  MoveL 6800 to (459.4, 541.64, 120) mm, rotated rx -180 ry 0 rz 160 deg; joints [12.499, 54.474, 8.674, -144.472, 67.608, 164.783]
  Set speed (16.1 mm/s)
  Call Extruder(646.01454)
  MoveL 6801 to (458.56, 540.8, 120) mm, rotated rx 180 ry 0 rz 160 deg; joints [12.412, 54.338, 8.962, -144.599, 67.708, 164.913]
  Set speed (16.1 mm/s)
  Call Extruder(649.31213)
  MoveL 6802 to (457.9, 540.12, 120) mm, rotated rx 180 ry 0 rz 160 deg; joints [12.341, 54.231, 9.187, -144.701, 67.786, 165.015]
  Set speed (16.1 mm/s)
  Call Extruder(654.34970)
  MoveL 6803 to (456.92, 539.07, 120) mm, rotated rx 180 ry 0 rz 160 deg; joints [12.227, 54.071, 9.524, -144.861, 67.902, 165.17]
  Set speed (16.1 mm/s)
  Call Extruder(658.51823)
  MoveL 6804 to (456.13, 538.18, 120) mm, rotated rx 180 ry 0 rz 160 deg; joints [12.13, 53.942, 9.797, -144.996, 67.995, 165.297]
  Set speed (16.1 mm/s)
  Call Extruder(662.65319)
  MoveL 6805 to (455.36, 537.28, 120) mm, rotated rx 180 ry 0 rz 160 deg; joints [12.031, 53.815, 10.064, -145.132, 68.085, 165.422]
  Set speed (16.1 mm/s)
  Call Extruder(666.83023)
  MoveL 6806 to (454.61, 536.36, 120) mm, rotated rx -180 ry 0 rz 160 deg; joints [11.927, 53.691, 10.328, -145.272, 68.173, 165.548]
  Call Extruder(670.95263)
  MoveL 6807 to (453.88, 535.43, 120) mm, rotated rx 180 ry 0 rz 160 deg; joints [11.822, 53.57, 10.582, -145.412, 68.257, 165.671]
  Set speed (16.1 mm/s)
  Call Extruder(675.12873)
  MoveL 6808 to (453.16, 534.48, 120) mm, rotated rx 180 ry 0 rz 160 deg; joints [11.713, 53.451, 10.836, -145.556, 68.34, 165.795]
  Set speed (16.1 mm/s)
  Call Extruder(679.32869)
  MoveL 6809 to (452.46, 533.5, 120) mm, rotated rx 180 ry 0 rz 160 deg; joints [11.599, 53.333, 11.084, -145.704, 68.421, 165.918]
  Set speed (16.1 mm/s)
  Call Extruder(683.43317)
  MoveL 6810 to (451.8, 532.54, 120) mm, rotated rx -180 ry 0 rz 160 deg; joints [11.485, 53.221, 11.321, -145.851, 68.497, 166.037]
  Set speed (16.1 mm/s)
  Call Extruder(686.86357)
  MoveL 6811 to (451.25, 531.72, 120) mm, rotated rx 180 ry 0 rz 160 deg; joints [11.388, 53.13, 11.516, -145.975, 68.558, 166.136]
  Set speed (16.1 mm/s)
  Call Extruder(691.76365)
  MoveL 6812 to (450.5, 530.53, 120) mm, rotated rx -180 ry 0 rz 160 deg; joints [11.246, 53.002, 11.786, -146.154, 68.643, 166.276]
  Set speed (16.1 mm/s)
  Call Extruder(695.89083)
  MoveL 6813 to (449.89, 529.52, 120) mm, rotated rx -180 ry 0 rz 160 deg; joints [11.123, 52.898, 12.007, -146.308, 68.711, 166.393]
  Set speed (16.1 mm/s)
  Call Extruder(700.22200)
  MoveL 6814 to (449.28, 528.45, 120) mm, rotated rx -180 ry 0 rz 160 deg; joints [10.991, 52.792, 12.233, -146.471, 68.78, 166.513]
  Set speed (16.1 mm/s)
  Call Extruder(704.20056)
  MoveL 6815 to (448.73, 527.46, 120) mm, rotated rx 180 ry 0 rz 160 deg; joints [10.868, 52.697, 12.434, -146.623, 68.84, 166.623]
  Set speed (16.1 mm/s)
  Call Extruder(708.45243)
  MoveL 6816 to (448.17, 526.38, 120) mm, rotated rx 180 ry 0 rz 160 deg; joints [10.733, 52.599, 12.643, -146.787, 68.902, 166.739]
  Set speed (16.1 mm/s)
  Call Extruder(712.70917)
  MoveL 6817 to (447.63, 525.29, 120) mm, rotated rx 180 ry 0 rz 160 deg; joints [10.595, 52.504, 12.846, -146.953, 68.961, 166.853]
  Call Extruder(720.90812)
  MoveL 6818 to (446.65, 523.16, 120) mm, rotated rx -180 ry 0 rz 160 deg; joints [10.323, 52.329, 13.218, -147.278, 69.065, 167.07]
  Set speed (16.1 mm/s)
  Call Extruder(729.11713)
  MoveL 6819 to (445.76, 520.99, 120) mm, rotated rx -180 ry 0 rz 160 deg; joints [10.041, 52.167, 13.564, -147.611, 69.157, 167.281]
  Set speed (16.1 mm/s)
  Call Extruder(733.49814)
  MoveL 6820 to (445.33, 519.82, 120) mm, rotated rx 180 ry 0 rz 160 deg; joints [9.886, 52.086, 13.737, -147.79, 69.201, 167.391]
  Call Extruder(737.53315)
  MoveL 6821 to (444.94, 518.73, 120) mm, rotated rx 180 ry 0 rz 160 deg; joints [9.743, 52.014, 13.892, -147.957, 69.24, 167.491]
  Set speed (16.1 mm/s)
  Call Extruder(741.86367)
  MoveL 6822 to (444.56, 517.56, 120) mm, rotated rx 180 ry 0 rz 160 deg; joints [9.586, 51.94, 14.049, -148.138, 69.277, 167.596]
  Call Extruder(745.89010)
  MoveL 6823 to (444.22, 516.46, 120) mm, rotated rx 180 ry 0 rz 160 deg; joints [9.439, 51.874, 14.191, -148.306, 69.309, 167.693]
  Set speed (16.1 mm/s)
  Call Extruder(754.18387)
  MoveL 6824 to (443.6, 514.17, 120) mm, rotated rx -180 ry 0 rz 160 deg; joints [9.129, 51.748, 14.459, -148.658, 69.366, 167.887]
  Set speed (16.1 mm/s)
  Call Extruder(757.85337)
  MoveL 6825 to (443.35, 513.15, 120) mm, rotated rx -180 ry 0 rz 160 deg; joints [8.989, 51.698, 14.568, -148.815, 69.386, 167.971]
  Set speed (16.1 mm/s)
  Call Extruder(763.31257)
  MoveL 6826 to (443.02, 511.63, 120) mm, rotated rx -180 ry 0 rz 160 deg; joints [8.78, 51.626, 14.722, -149.05, 69.413, 168.093]
  Set speed (16.1 mm/s)
  Call Extruder(771.04723)
  MoveL 6827 to (442.62, 509.46, 120) mm, rotated rx -180 ry 0 rz 160 deg; joints [8.478, 51.534, 14.918, -149.385, 69.441, 168.261]
  Set speed (16.1 mm/s)
  Call Extruder(779.38114)
  MoveL 6828 to (442.28, 507.1, 120) mm, rotated rx -180 ry 0 rz 160 deg; joints [8.148, 51.449, 15.102, -149.75, 69.459, 168.435]
  Call Extruder(787.70369)
  MoveL 6829 to (442.04, 504.74, 120) mm, rotated rx 180 ry 0 rz 160 deg; joints [7.813, 51.377, 15.255, -150.116, 69.463, 168.602]
  Call Extruder(795.81403)
  MoveL 6830 to (441.89, 502.42, 120) mm, rotated rx 180 ry 0 rz 160 deg; joints [7.483, 51.32, 15.377, -150.473, 69.455, 168.758]
  Call Extruder(804.25342)
  MoveL 6831 to (441.84, 500.01, 120) mm, rotated rx -180 ry 0 rz 160 deg; joints [7.136, 51.275, 15.474, -150.846, 69.433, 168.912]
  Set speed (16.1 mm/s)
  Call Extruder(811.82598)
  MoveL 6832 to (441.88, 497.85, 120) mm, rotated rx 180 ry 0 rz 160 deg; joints [6.823, 51.247, 15.534, -151.18, 69.401, 169.044]
  Call Extruder(819.14286)
  MoveL 6833 to (442, 495.76, 120) mm, rotated rx -180 ry 0 rz 160 deg; joints [6.52, 51.231, 15.568, -151.502, 69.36, 169.166]
  Call Extruder(826.71033)
  MoveL 6834 to (442.19, 493.61, 120) mm, rotated rx 180 ry 0 rz 160 deg; joints [6.205, 51.226, 15.58, -151.833, 69.307, 169.286]
  Set speed (16.1 mm/s)
  Call Extruder(834.19803)
  MoveL 6835 to (442.47, 491.48, 120) mm, rotated rx 180 ry 0 rz 160 deg; joints [5.894, 51.232, 15.566, -152.159, 69.242, 169.398]
  Call Extruder(841.79303)
  MoveL 6836 to (442.83, 489.34, 120) mm, rotated rx -180 ry 0 rz 160 deg; joints [5.578, 51.25, 15.528, -152.487, 69.167, 169.505]
  Set speed (16.1 mm/s)
  Call Extruder(849.45555)
  MoveL 6837 to (443.27, 487.19, 120) mm, rotated rx 180 ry 0 rz 160 deg; joints [5.262, 51.28, 15.464, -152.814, 69.079, 169.607]
  Call Extruder(856.66940)
  MoveL 6838 to (443.76, 485.19, 120) mm, rotated rx 180 ry 0 rz 160 deg; joints [4.966, 51.319, 15.381, -153.119, 68.986, 169.697]
  Set speed (16.1 mm/s)
  Call Extruder(864.15213)
  MoveL 6839 to (444.34, 483.13, 120) mm, rotated rx 180 ry 0 rz 160 deg; joints [4.661, 51.37, 15.27, -153.43, 68.879, 169.784]
  Set speed (16.1 mm/s)
  Call Extruder(871.56534)
  MoveL 6840 to (444.99, 481.12, 120) mm, rotated rx -180 ry 0 rz 160 deg; joints [4.362, 51.432, 15.137, -153.733, 68.763, 169.864]
  Set speed (16.1 mm/s)
  Call Extruder(879.13739)
  MoveL 6841 to (445.73, 479.08, 120) mm, rotated rx -180 ry 0 rz 160 deg; joints [4.06, 51.506, 14.978, -154.037, 68.633, 169.94]
  Set speed (16.1 mm/s)
  Call Extruder(885.78650)
  MoveL 6842 to (446.45, 477.32, 120) mm, rotated rx 180 ry 0 rz 160 deg; joints [3.799, 51.581, 14.818, -154.299, 68.511, 170.001]
  Call Extruder(894.03037)
  MoveL 6843 to (447.41, 475.17, 120) mm, rotated rx 180 ry 0 rz 160 deg; joints [3.481, 51.686, 14.593, -154.616, 68.348, 170.069]
  Set speed (16.1 mm/s)
  Call Extruder(901.71326)
  MoveL 6844 to (448.39, 473.2, 120) mm, rotated rx -180 ry 0 rz 160 deg; joints [3.19, 51.795, 14.359, -154.903, 68.185, 170.127]
  Set speed (16.1 mm/s)
  Call Extruder(909.01008)
  MoveL 6845 to (449.38, 471.37, 120) mm, rotated rx 180 ry 0 rz 160 deg; joints [2.919, 51.909, 14.115, -155.168, 68.021, 170.175]
  Set speed (16.1 mm/s)
  Call Extruder(916.69414)
  MoveL 6846 to (450.49, 469.48, 120) mm, rotated rx 180 ry 0 rz 160 deg; joints [2.64, 52.04, 13.835, -155.439, 67.838, 170.219]
  Call Extruder(924.08438)
  MoveL 6847 to (451.64, 467.7, 120) mm, rotated rx 180 ry 0 rz 160 deg; joints [2.379, 52.177, 13.544, -155.691, 67.653, 170.255]
  Set speed (16.1 mm/s)
  Call Extruder(931.57807)
  MoveL 6848 to (452.86, 465.94, 120) mm, rotated rx 180 ry 0 rz 160 deg; joints [2.122, 52.325, 13.227, -155.937, 67.456, 170.285]
  Call Extruder(939.16479)
  MoveL 6849 to (454.16, 464.21, 120) mm, rotated rx -180 ry 0 rz 160 deg; joints [1.869, 52.486, 12.884, -156.177, 67.247, 170.309]
  Set speed (16.1 mm/s)
  Call Extruder(946.56366)
  MoveL 6850 to (455.49, 462.57, 120) mm, rotated rx 180 ry 0 rz 160 deg; joints [1.631, 52.652, 12.53, -156.4, 67.035, 170.326]
  Call Extruder(954.04593)
  MoveL 6851 to (456.9, 460.96, 120) mm, rotated rx 180 ry 0 rz 160 deg; joints [1.398, 52.831, 12.151, -156.615, 66.812, 170.337]
  Set speed (16.1 mm/s)
  Call Extruder(961.81892)
  MoveL 6852 to (458.42, 459.34, 120) mm, rotated rx -180 ry 0 rz 160 deg; joints [1.166, 53.026, 11.737, -156.827, 66.571, 170.341]
  Call Extruder(968.91322)
  MoveL 6853 to (459.87, 457.91, 120) mm, rotated rx 180 ry 0 rz 160 deg; joints [0.962, 53.212, 11.341, -157.01, 66.344, 170.339]
  Call Extruder(976.52373)
  MoveL 6854 to (461.47, 456.44, 120) mm, rotated rx 180 ry 0 rz 160 deg; joints [0.753, 53.422, 10.897, -157.195, 66.093, 170.33]
  Set speed (16.1 mm/s)
  Call Extruder(984.09802)
  MoveL 6855 to (463.12, 455.04, 120) mm, rotated rx -180 ry 0 rz 160 deg; joints [0.555, 53.639, 10.437, -157.367, 65.836, 170.315]
  Set speed (16.1 mm/s)
  Call Extruder(991.96002)
  MoveL 6856 to (464.88, 453.64, 120) mm, rotated rx 180 ry 0 rz 160 deg; joints [0.36, 53.874, 9.94, -157.533, 65.562, 170.291]
  Call Extruder(999.08695)
  MoveL 6857 to (466.52, 452.44, 120) mm, rotated rx -180 ry 0 rz 160 deg; joints [0.193, 54.095, 9.474, -157.671, 65.306, 170.264]
  Set speed (16.1 mm/s)
  Call Extruder(1006.48210)
  MoveL 6858 to (468.27, 451.26, 120) mm, rotated rx 180 ry 0 rz 160 deg; joints [0.03, 54.332, 8.974, -157.802, 65.036, 170.229]
  Set speed (16.1 mm/s)
  Call Extruder(1014.06845)
  MoveL 6859 to (470.11, 450.11, 120) mm, rotated rx 180 ry 0 rz 160 deg; joints [-0.127, 54.583, 8.445, -157.924, 64.752, 170.186]
  Set speed (16.1 mm/s)
  Call Extruder(1021.55574)
  MoveL 6860 to (471.97, 449.04, 120) mm, rotated rx 180 ry 0 rz 160 deg; joints [-0.272, 54.838, 7.909, -158.032, 64.466, 170.136]
  Set speed (16.1 mm/s)
  Call Extruder(1029.94377)
  MoveL 6861 to (474.09, 447.93, 120) mm, rotated rx 180 ry 0 rz 160 deg; joints [-0.421, 55.133, 7.291, -158.137, 64.14, 170.073]
  Set speed (16.1 mm/s)
  Call Extruder(1036.55206)
  MoveL 6862 to (475.8, 447.12, 120) mm, rotated rx 180 ry 0 rz 160 deg; joints [-0.529, 55.371, 6.791, -158.207, 63.879, 170.017]
  Set speed (16.1 mm/s)
  Call Extruder(1044.03826)
  MoveL 6863 to (477.76, 446.27, 120) mm, rotated rx -180 ry 0 rz 160 deg; joints [-0.641, 55.647, 6.213, -158.275, 63.579, 169.946]
  Set speed (16.1 mm/s)
  Call Extruder(1051.32870)
  MoveL 6864 to (479.69, 445.5, 120) mm, rotated rx -180 ry 0 rz 160 deg; joints [-0.74, 55.923, 5.638, -158.329, 63.283, 169.871]
  Call Extruder(1059.02695)
  MoveL 6865 to (481.77, 444.77, 120) mm, rotated rx -180 ry 0 rz 160 deg; joints [-0.833, 56.219, 5.018, -158.371, 62.967, 169.784]
  Call Extruder(1066.47364)
  MoveL 6866 to (483.8, 444.14, 120) mm, rotated rx 180 ry 0 rz 160 deg; joints [-0.913, 56.512, 4.407, -158.399, 62.657, 169.693]
  Call Extruder(1073.74383)
  MoveL 6867 to (485.81, 443.6, 120) mm, rotated rx -180 ry 0 rz 160 deg; joints [-0.98, 56.804, 3.801, -158.413, 62.352, 169.596]
  Set speed (16.1 mm/s)
  Call Extruder(1081.50301)
  MoveL 6868 to (487.97, 443.1, 120) mm, rotated rx 180 ry 0 rz 160 deg; joints [-1.04, 57.12, 3.144, -158.414, 62.024, 169.486]
  Call Extruder(1088.89317)
  MoveL 6869 to (490.05, 442.7, 120) mm, rotated rx 180 ry 0 rz 160 deg; joints [-1.088, 57.426, 2.51, -158.403, 61.71, 169.374]
  Set speed (16.1 mm/s)
  Call Extruder(1096.03300)
  MoveL 6870 to (492.06, 442.39, 120) mm, rotated rx -180 ry 0 rz 160 deg; joints [-1.124, 57.725, 1.889, -158.379, 61.405, 169.258]
  Set speed (16.1 mm/s)
  Call Extruder(1103.71272)
  MoveL 6871 to (494.24, 442.13, 120) mm, rotated rx 180 ry 0 rz 160 deg; joints [-1.151, 58.051, 1.214, -158.339, 61.075, 169.126]
  Set speed (16.1 mm/s)
  Call Extruder(1111.28299)
  MoveL 6872 to (496.4, 441.95, 120) mm, rotated rx 180 ry 0 rz 160 deg; joints [-1.168, 58.377, 0.541, -158.286, 60.749, 168.989]
  Set speed (16.1 mm/s)
  Call Extruder(1118.95323)
  MoveL 6873 to (498.59, 441.86, 120) mm, rotated rx -180 ry 0 rz 160 deg; joints [-1.175, 58.71, -0.147, -158.22, 60.419, 168.842]
  Set speed (16.1 mm/s)
  Call Extruder(1126.35629)
  MoveL 6874 to (500.71, 441.85, 120) mm, rotated rx -180 ry 0 rz 160 deg; joints [-1.171, 59.035, -0.816, -158.142, 60.1, 168.692]
  Call Extruder(1133.91680)
  MoveL 6875 to (502.87, 441.91, 120) mm, rotated rx -180 ry 0 rz 160 deg; joints [-1.157, 59.369, -1.504, -158.05, 59.774, 168.532]
  Call Extruder(1141.32935)
  MoveL 6876 to (504.98, 442.06, 120) mm, rotated rx 180 ry 0 rz 160 deg; joints [-1.133, 59.699, -2.182, -157.947, 59.456, 168.367]
  Set speed (16.1 mm/s)
  Call Extruder(1148.64149)
  MoveL 6877 to (507.06, 442.27, 120) mm, rotated rx -180 ry 0 rz 160 deg; joints [-1.101, 60.026, -2.853, -157.833, 59.144, 168.197]
  Set speed (16.1 mm/s)
  Call Extruder(1156.31820)
  MoveL 6878 to (509.23, 442.58, 120) mm, rotated rx -180 ry 0 rz 160 deg; joints [-1.057, 60.371, -3.56, -157.701, 58.818, 168.012]
  Set speed (16.1 mm/s)
  Call Extruder(1163.87434)
  MoveL 6879 to (511.36, 442.96, 120) mm, rotated rx 180 ry 0 rz 160 deg; joints [-1.005, 60.711, -4.256, -157.559, 58.5, 167.822]
  Set speed (16.1 mm/s)
  Call Extruder(1171.29769)
  MoveL 6880 to (513.43, 443.41, 120) mm, rotated rx 180 ry 0 rz 160 deg; joints [-0.945, 61.046, -4.941, -157.407, 58.189, 167.628]
  Set speed (16.1 mm/s)
  Call Extruder(1178.67571)
  MoveL 6881 to (515.47, 443.94, 120) mm, rotated rx -180 ry 0 rz 160 deg; joints [-0.876, 61.38, -5.622, -157.244, 57.884, 167.429]
  Set speed (16.1 mm/s)
  Call Extruder(1186.11275)
  MoveL 6882 to (517.51, 444.54, 120) mm, rotated rx 180 ry 0 rz 160 deg; joints [-0.798, 61.715, -6.306, -157.068, 57.58, 167.221]
  Call Extruder(1193.83773)
  MoveL 6883 to (519.6, 445.25, 120) mm, rotated rx -180 ry 0 rz 160 deg; joints [-0.708, 62.063, -7.015, -156.874, 57.268, 166.997]
  Set speed (16.1 mm/s)
  Call Extruder(1201.22298)
  MoveL 6884 to (521.58, 445.99, 120) mm, rotated rx -180 ry 0 rz 160 deg; joints [-0.614, 62.395, -7.689, -156.678, 56.974, 166.777]
  Set speed (16.1 mm/s)
  Call Extruder(1208.63995)
  MoveL 6885 to (523.53, 446.82, 120) mm, rotated rx -180 ry 0 rz 160 deg; joints [-0.512, 62.726, -8.363, -156.47, 56.683, 166.549]
  Set speed (16.1 mm/s)
  Call Extruder(1215.26606)
  MoveL 6886 to (525.25, 447.61, 120) mm, rotated rx -180 ry 0 rz 160 deg; joints [-0.414, 63.021, -8.961, -156.277, 56.428, 166.341]
  Set speed (16.1 mm/s)
  Call Extruder(1223.71389)
  MoveL 6887 to (527.4, 448.7, 120) mm, rotated rx -180 ry 0 rz 160 deg; joints [-0.281, 63.393, -9.716, -156.017, 56.11, 166.069]
  Set speed (16.1 mm/s)
  Call Extruder(1231.29077)
  MoveL 6888 to (529.3, 449.76, 120) mm, rotated rx 180 ry 0 rz 160 deg; joints [-0.153, 63.725, -10.387, -155.774, 55.831, 165.818]
  Set speed (16.1 mm/s)
  Call Extruder(1238.69731)
  MoveL 6889 to (531.11, 450.86, 120) mm, rotated rx 180 ry 0 rz 160 deg; joints [-0.022, 64.045, -11.035, -155.528, 55.565, 165.567]
  Set speed (16.1 mm/s)
  Call Extruder(1246.28249)
  MoveL 6890 to (532.92, 452.06, 120) mm, rotated rx 180 ry 0 rz 160 deg; joints [0.12, 64.369, -11.69, -155.266, 55.3, 165.305]
  Set speed (16.1 mm/s)
  Call Extruder(1253.66351)
  MoveL 6891 to (534.63, 453.28, 120) mm, rotated rx 180 ry 0 rz 160 deg; joints [0.265, 64.681, -12.319, -155.003, 55.049, 165.045]
  Call Extruder(1261.15428)
  MoveL 6892 to (536.33, 454.59, 120) mm, rotated rx 180 ry 0 rz 160 deg; joints [0.418, 64.992, -12.946, -154.728, 54.803, 164.778]
  Set speed (16.1 mm/s)
  Call Extruder(1268.66408)
  MoveL 6893 to (537.98, 455.96, 120) mm, rotated rx 180 ry 0 rz 160 deg; joints [0.578, 65.298, -13.563, -154.444, 54.564, 164.505]
  Set speed (16.1 mm/s)
  Call Extruder(1276.05790)
  MoveL 6894 to (539.55, 457.37, 120) mm, rotated rx 180 ry 0 rz 160 deg; joints [0.741, 65.594, -14.16, -154.158, 54.338, 164.233]
  Set speed (16.1 mm/s)
  Call Extruder(1283.76960)
  MoveL 6895 to (541.14, 458.9, 120) mm, rotated rx 180 ry 0 rz 160 deg; joints [0.917, 65.897, -14.768, -153.853, 54.112, 163.945]
  Call Extruder(1287.76845)
  MoveL 6896 to (541.94, 459.71, 120) mm, rotated rx 180 ry 0 rz 160 deg; joints [1.011, 66.051, -15.078, -153.692, 53.998, 163.795]
  Set speed (16.1 mm/s)
  Call Extruder(1291.96467)
  MoveL 6897 to (542.76, 460.58, 120) mm, rotated rx 180 ry 0 rz 160 deg; joints [1.111, 66.211, -15.398, -153.521, 53.882, 163.637]
  Set speed (16.1 mm/s)
  Call Extruder(1296.08175)
  MoveL 6898 to (543.55, 461.46, 120) mm, rotated rx -180 ry 0 rz 160 deg; joints [1.211, 66.364, -15.707, -153.352, 53.771, 163.481]
  Set speed (16.1 mm/s)
  Call Extruder(1300.19670)
  MoveL 6899 to (544.32, 462.35, 120) mm, rotated rx -180 ry 0 rz 160 deg; joints [1.312, 66.517, -16.012, -153.181, 53.664, 163.324]
  Set speed (16.1 mm/s)
  Call Extruder(1304.40956)
  MoveL 6900 to (545.09, 463.27, 120) mm, rotated rx 180 ry 0 rz 160 deg; joints [1.417, 66.67, -16.319, -153.005, 53.557, 163.164]
  Call Extruder(1308.57141)
  MoveL 6901 to (545.83, 464.2, 120) mm, rotated rx -180 ry 0 rz 160 deg; joints [1.522, 66.818, -16.617, -152.829, 53.454, 163.004]
  Call Extruder(1312.66863)
  MoveL 6902 to (546.55, 465.13, 120) mm, rotated rx 180 ry 0 rz 160 deg; joints [1.628, 66.962, -16.905, -152.654, 53.357, 162.847]
  Set speed (16.1 mm/s)
  Call Extruder(1316.96653)
  MoveL 6903 to (547.27, 466.12, 120) mm, rotated rx -180 ry 0 rz 160 deg; joints [1.74, 67.11, -17.202, -152.47, 53.258, 162.682]
  Call Extruder(1321.10983)
  MoveL 6904 to (547.95, 467.09, 120) mm, rotated rx 180 ry 0 rz 160 deg; joints [1.849, 67.25, -17.482, -152.291, 53.167, 162.523]
  Call Extruder(1325.92423)
  MoveL 6905 to (548.72, 468.24, 120) mm, rotated rx -180 ry 0 rz 160 deg; joints [1.978, 67.409, -17.801, -152.082, 53.064, 162.338]
  Call Extruder(1329.43388)
  MoveL 6906 to (549.26, 469.08, 120) mm, rotated rx -180 ry 0 rz 160 deg; joints [2.073, 67.522, -18.027, -151.929, 52.993, 162.203]
  Set speed (16.1 mm/s)
  Call Extruder(1333.55402)
  MoveL 6907 to (549.87, 470.09, 120) mm, rotated rx -180 ry 0 rz 160 deg; joints [2.185, 67.653, -18.288, -151.748, 52.913, 162.045]
  Set speed (16.1 mm/s)
  Call Extruder(1337.62936)
  MoveL 6908 to (550.46, 471.09, 120) mm, rotated rx -180 ry 0 rz 160 deg; joints [2.297, 67.779, -18.54, -151.569, 52.837, 161.89]
  Set speed (16.1 mm/s)
  Call Extruder(1341.78518)
  MoveL 6909 to (551.04, 472.13, 120) mm, rotated rx 180 ry 0 rz 160 deg; joints [2.413, 67.904, -18.791, -151.385, 52.763, 161.731]
  Set speed (16.1 mm/s)
  Call Extruder(1345.99468)
  MoveL 6910 to (551.61, 473.19, 120) mm, rotated rx -180 ry 0 rz 160 deg; joints [2.532, 68.028, -19.038, -151.199, 52.692, 161.571]
  Set speed (16.1 mm/s)
  Call Extruder(1350.18264)
  MoveL 6911 to (552.15, 474.26, 120) mm, rotated rx -180 ry 0 rz 160 deg; joints [2.651, 68.148, -19.277, -151.013, 52.625, 161.412]
  Set speed (16.1 mm/s)
  Call Extruder(1354.31072)
  MoveL 6912 to (552.66, 475.32, 120) mm, rotated rx 180 ry 0 rz 160 deg; joints [2.769, 68.262, -19.505, -150.829, 52.563, 161.257]
  Set speed (16.1 mm/s)
  Call Extruder(1358.53123)
  MoveL 6913 to (553.16, 476.42, 120) mm, rotated rx 180 ry 0 rz 160 deg; joints [2.891, 68.375, -19.731, -150.642, 52.504, 161.099]
  Call Extruder(1366.91580)
  MoveL 6914 to (554.09, 478.63, 120) mm, rotated rx 180 ry 0 rz 160 deg; joints [3.137, 68.59, -20.16, -150.268, 52.399, 160.787]
  Set speed (16.1 mm/s)
  Call Extruder(1375.14529)
  MoveL 6915 to (554.91, 480.83, 120) mm, rotated rx -180 ry 0 rz 160 deg; joints [3.381, 68.786, -20.55, -149.901, 52.311, 160.487]
  Set speed (16.1 mm/s)
  Call Extruder(1379.37701)
  MoveL 6916 to (555.29, 481.98, 120) mm, rotated rx 180 ry 0 rz 160 deg; joints [3.509, 68.88, -20.737, -149.714, 52.273, 160.335]
  Call Extruder(1383.73199)
  MoveL 6917 to (555.67, 483.16, 120) mm, rotated rx 180 ry 0 rz 160 deg; joints [3.64, 68.974, -20.925, -149.521, 52.237, 160.179]
  Call Extruder(1387.70261)
  MoveL 6918 to (555.98, 484.25, 120) mm, rotated rx -180 ry 0 rz 160 deg; joints [3.761, 69.054, -21.085, -149.346, 52.209, 160.04]
  Set speed (16.1 mm/s)
  Call Extruder(1391.64358)
  MoveL 6919 to (556.28, 485.34, 120) mm, rotated rx 180 ry 0 rz 160 deg; joints [3.881, 69.132, -21.24, -149.172, 52.184, 159.902]
  Set speed (16.1 mm/s)
  Call Extruder(1400.07126)
  MoveL 6920 to (556.84, 487.68, 120) mm, rotated rx 180 ry 0 rz 160 deg; joints [4.141, 69.285, -21.544, -148.803, 52.144, 159.614]
  Set speed (16.1 mm/s)
  Call Extruder(1408.49387)
  MoveL 6921 to (557.3, 490.05, 120) mm, rotated rx 180 ry 0 rz 160 deg; joints [4.403, 69.42, -21.813, -148.438, 52.122, 159.335]
  Set speed (16.1 mm/s)
  Call Extruder(1416.73608)
  MoveL 6922 to (557.65, 492.37, 120) mm, rotated rx 180 ry 0 rz 160 deg; joints [4.661, 69.535, -22.041, -148.085, 52.117, 159.072]
  Set speed (16.1 mm/s)
  Call Extruder(1425.23980)
  MoveL 6923 to (557.92, 494.79, 120) mm, rotated rx 180 ry 0 rz 160 deg; joints [4.93, 69.635, -22.242, -147.727, 52.129, 158.81]
  Set speed (16.1 mm/s)
  Call Extruder(1433.45629)
  MoveL 6924 to (558.09, 497.13, 120) mm, rotated rx -180 ry 0 rz 160 deg; joints [5.191, 69.715, -22.399, -147.386, 52.158, 158.567]
  Set speed (16.1 mm/s)
  Call Extruder(1441.77748)
  MoveL 6925 to (558.16, 499.51, 120) mm, rotated rx 180 ry 0 rz 160 deg; joints [5.456, 69.777, -22.524, -147.047, 52.203, 158.333]
  Set speed (16.1 mm/s)
  Call Extruder(1449.93682)
  MoveL 6926 to (558.13, 501.85, 120) mm, rotated rx 180 ry 0 rz 160 deg; joints [5.718, 69.821, -22.61, -146.722, 52.265, 158.116]
  Set speed (16.1 mm/s)
  Call Extruder(1458.38997)
  MoveL 6927 to (558, 504.26, 120) mm, rotated rx 180 ry 0 rz 160 deg; joints [5.989, 69.846, -22.661, -146.393, 52.345, 157.903]
  Set speed (16.1 mm/s)
  Call Extruder(1466.71982)
  MoveL 6928 to (557.78, 506.63, 120) mm, rotated rx 180 ry 0 rz 160 deg; joints [6.256, 69.853, -22.674, -146.078, 52.441, 157.708]
  Set speed (16.1 mm/s)
  Call Extruder(1475.15035)
  MoveL 6929 to (557.45, 509.02, 120) mm, rotated rx -180 ry 0 rz 160 deg; joints [6.527, 69.841, -22.65, -145.768, 52.554, 157.525]
  Set speed (16.1 mm/s)
  Call Extruder(1483.23849)
  MoveL 6930 to (557.05, 511.3, 120) mm, rotated rx -180 ry 0 rz 160 deg; joints [6.787, 69.811, -22.591, -145.479, 52.677, 157.362]
  Set speed (16.1 mm/s)
  Call Extruder(1491.85094)
  MoveL 6931 to (556.52, 513.71, 120) mm, rotated rx 180 ry 0 rz 160 deg; joints [7.062, 69.76, -22.49, -145.181, 52.825, 157.205]
  Set speed (16.1 mm/s)
  Call Extruder(1499.78968)
  MoveL 6932 to (555.94, 515.9, 120) mm, rotated rx 180 ry 0 rz 160 deg; joints [7.315, 69.696, -22.362, -144.916, 52.976, 157.074]
  Set speed (16.1 mm/s)
  Call Extruder(1508.42581)
  MoveL 6933 to (555.22, 518.26, 120) mm, rotated rx 180 ry 0 rz 160 deg; joints [7.589, 69.607, -22.185, -144.639, 53.154, 156.948]
  Set speed (16.1 mm/s)
  Call Extruder(1516.59565)
  MoveL 6934 to (554.44, 520.46, 120) mm, rotated rx 180 ry 0 rz 160 deg; joints [7.847, 69.506, -21.983, -144.387, 53.337, 156.844]
  Set speed (16.1 mm/s)
  Call Extruder(1524.82299)
  MoveL 6935 to (553.57, 522.65, 120) mm, rotated rx -180 ry 0 rz 160 deg; joints [8.104, 69.387, -21.747, -144.143, 53.534, 156.754]
  Set speed (16.1 mm/s)
  Call Extruder(1533.21607)
  MoveL 6936 to (552.59, 524.84, 120) mm, rotated rx 180 ry 0 rz 160 deg; joints [8.365, 69.247, -21.469, -143.905, 53.749, 156.678]
  Set speed (16.1 mm/s)
  Call Extruder(1537.37064)
  MoveL 6937 to (552.07, 525.91, 120) mm, rotated rx -180 ry 0 rz 160 deg; joints [8.493, 69.171, -21.318, -143.792, 53.86, 156.647]
  Set speed (16.1 mm/s)
  Call Extruder(1543.51098)
  MoveL 6938 to (551.26, 527.47, 120) mm, rotated rx 180 ry 0 rz 160 deg; joints [8.681, 69.053, -21.083, -143.629, 54.029, 156.607]
  Set speed (16.2 mm/s)
  Call Extruder(1549.80649)
  MoveL 6939 to (550.39, 529.04, 120) mm, rotated rx 180 ry 0 rz 160 deg; joints [8.873, 68.921, -20.821, -143.468, 54.211, 156.576]
  Set speed (16.1 mm/s)
  Call Extruder(1553.96982)
  MoveL 6940 to (549.78, 530.07, 120) mm, rotated rx -180 ry 0 rz 160 deg; joints [8.998, 68.83, -20.639, -143.365, 54.333, 156.56]
  Call Extruder(1558.22289)
  MoveL 6941 to (549.14, 531.1, 120) mm, rotated rx -180 ry 0 rz 160 deg; joints [9.125, 68.732, -20.443, -143.264, 54.462, 156.548]
  Set speed (16.1 mm/s)
  Call Extruder(1562.31252)
  MoveL 6942 to (548.51, 532.09, 120) mm, rotated rx 180 ry 0 rz 160 deg; joints [9.247, 68.635, -20.249, -143.168, 54.588, 156.54]
  Set speed (16.1 mm/s)
  Call Extruder(1566.58984)
  MoveL 6943 to (547.82, 533.1, 120) mm, rotated rx 180 ry 0 rz 160 deg; joints [9.373, 68.529, -20.038, -143.071, 54.722, 156.535]
  Set speed (16.1 mm/s)
  Call Extruder(1571.39278)
  MoveL 6944 to (547.02, 534.22, 120) mm, rotated rx -180 ry 0 rz 160 deg; joints [9.513, 68.405, -19.79, -142.966, 54.877, 156.535]
  Call Extruder(0.00000)
  Call Extruder(3.43739)
  MoveL 6945 to (546.44, 535.01, 120) mm, rotated rx 180 ry 0 rz 160 deg; joints [9.613, 68.314, -19.609, -142.892, 54.989, 156.537]
  Set speed (16.1 mm/s)
  Call Extruder(8.16081)
  MoveL 6946 to (545.62, 536.08, 120) mm, rotated rx -180 ry 0 rz 160 deg; joints [9.749, 68.185, -19.351, -142.794, 55.146, 156.545]
  Set speed (16.1 mm/s)
  Call Extruder(11.80532)
  MoveL 6947 to (544.96, 536.89, 120) mm, rotated rx 180 ry 0 rz 160 deg; joints [9.853, 68.082, -19.145, -142.721, 55.269, 156.554]
  Set speed (16.1 mm/s)
  Call Extruder(15.90025)
  MoveL 6948 to (544.21, 537.78, 120) mm, rotated rx 180 ry 0 rz 160 deg; joints [9.969, 67.963, -18.907, -142.642, 55.409, 156.569]
  Set speed (16.1 mm/s)
  Call Extruder(20.03659)
  MoveL 6949 to (543.43, 538.68, 120) mm, rotated rx 180 ry 0 rz 160 deg; joints [10.085, 67.839, -18.661, -142.564, 55.553, 156.586]
  Set speed (16.1 mm/s)
  Call Extruder(24.30870)
  MoveL 6950 to (542.61, 539.58, 120) mm, rotated rx -180 ry 0 rz 160 deg; joints [10.204, 67.709, -18.4, -142.487, 55.704, 156.608]
  Set speed (16.1 mm/s)
  Call Extruder(28.36774)
  MoveL 6951 to (541.81, 540.42, 120) mm, rotated rx 180 ry 0 rz 160 deg; joints [10.315, 67.581, -18.145, -142.416, 55.849, 156.632]
  Set speed (16.1 mm/s)
  Call Extruder(32.58030)
  MoveL 6952 to (540.97, 541.28, 120) mm, rotated rx -180 ry 0 rz 160 deg; joints [10.429, 67.446, -17.875, -142.345, 56.001, 156.661]
  Set speed (16.1 mm/s)
  Call Extruder(36.77160)
  MoveL 6953 to (540.11, 542.12, 120) mm, rotated rx 180 ry 0 rz 160 deg; joints [10.542, 67.309, -17.601, -142.277, 56.155, 156.692]
  Set speed (16.1 mm/s)
  Call Extruder(40.84066)
  MoveL 6954 to (539.26, 542.91, 120) mm, rotated rx -180 ry 0 rz 160 deg; joints [10.65, 67.173, -17.328, -142.214, 56.305, 156.727]
  Set speed (16.1 mm/s)
  Call Extruder(44.99678)
  MoveL 6955 to (538.37, 543.7, 120) mm, rotated rx 180 ry 0 rz 160 deg; joints [10.758, 67.031, -17.043, -142.151, 56.461, 156.765]
  Set speed (16.1 mm/s)
  Call Extruder(49.25698)
  MoveL 6956 to (537.45, 544.49, 120) mm, rotated rx -180 ry 0 rz 160 deg; joints [10.868, 66.883, -16.746, -142.091, 56.622, 156.808]
  Set speed (16.1 mm/s)
  Call Extruder(53.34054)
  MoveL 6957 to (536.55, 545.24, 120) mm, rotated rx 180 ry 0 rz 160 deg; joints [10.973, 66.738, -16.457, -142.035, 56.777, 156.852]
  Set speed (16.1 mm/s)
  Call Extruder(57.63629)
  MoveL 6958 to (535.59, 546, 120) mm, rotated rx -180 ry 0 rz 160 deg; joints [11.081, 66.583, -16.146, -141.979, 56.942, 156.901]
  Set speed (16.1 mm/s)
  Call Extruder(61.65074)
  MoveL 6959 to (534.67, 546.69, 120) mm, rotated rx 180 ry 0 rz 160 deg; joints [11.18, 66.436, -15.85, -141.929, 57.098, 156.951]
  Set speed (16.1 mm/s)
  Call Extruder(65.84245)
  MoveL 6960 to (533.7, 547.4, 120) mm, rotated rx 180 ry 0 rz 160 deg; joints [11.282, 66.28, -15.538, -141.879, 57.261, 157.005]
  Set speed (16.1 mm/s)
  Call Extruder(69.96501)
  MoveL 6961 to (532.74, 548.07, 120) mm, rotated rx -180 ry 0 rz 160 deg; joints [11.381, 66.124, -15.225, -141.833, 57.423, 157.062]
  Set speed (16.1 mm/s)
  Call Extruder(74.19741)
  MoveL 6962 to (531.73, 548.74, 120) mm, rotated rx 180 ry 0 rz 160 deg; joints [11.481, 65.962, -14.899, -141.789, 57.591, 157.124]
  Call Extruder(78.26454)
  MoveL 6963 to (530.75, 549.37, 120) mm, rotated rx -180 ry 0 rz 160 deg; joints [11.576, 65.805, -14.582, -141.748, 57.753, 157.185]
  Set speed (16.1 mm/s)
  Call Extruder(82.50052)
  MoveL 6964 to (529.71, 550, 120) mm, rotated rx -180 ry 0 rz 160 deg; joints [11.672, 65.638, -14.247, -141.708, 57.922, 157.252]
  Set speed (16.1 mm/s)
  Call Extruder(86.66587)
  MoveL 6965 to (528.68, 550.59, 120) mm, rotated rx 180 ry 0 rz 160 deg; joints [11.765, 65.472, -13.913, -141.672, 58.09, 157.321]
  Set speed (16.1 mm/s)
  Call Extruder(93.50570)
  MoveL 6966 to (526.97, 551.53, 120) mm, rotated rx 180 ry 0 rz 160 deg; joints [11.914, 65.197, -13.359, -141.617, 58.366, 157.44]
  Set speed (16.1 mm/s)
  Call Extruder(99.11961)
  MoveL 6967 to (525.54, 552.25, 120) mm, rotated rx -180 ry 0 rz 160 deg; joints [12.033, 64.966, -12.895, -141.579, 58.595, 157.543]
  Set speed (16.1 mm/s)
  Call Extruder(103.28725)
  MoveL 6968 to (524.46, 552.76, 120) mm, rotated rx 180 ry 0 rz 160 deg; joints [12.118, 64.794, -12.546, -141.552, 58.765, 157.623]
  Set speed (16.1 mm/s)
  Call Extruder(111.55058)
  MoveL 6969 to (522.3, 553.72, 120) mm, rotated rx 180 ry 0 rz 160 deg; joints [12.283, 64.447, -11.847, -141.507, 59.103, 157.787]
  Set speed (16.1 mm/s)
  Call Extruder(115.82777)
  MoveL 6970 to (521.16, 554.17, 120) mm, rotated rx 180 ry 0 rz 160 deg; joints [12.364, 64.265, -11.479, -141.488, 59.279, 157.877]
  Set speed (16.1 mm/s)
  Call Extruder(120.02852)
  MoveL 6971 to (520.04, 554.59, 120) mm, rotated rx -180 ry 0 rz 160 deg; joints [12.442, 64.086, -11.117, -141.471, 59.452, 157.967]
  Set speed (16.1 mm/s)
  Call Extruder(124.24046)
  MoveL 6972 to (518.91, 554.99, 120) mm, rotated rx -180 ry 0 rz 160 deg; joints [12.518, 63.904, -10.749, -141.458, 59.626, 158.06]
  Set speed (16.1 mm/s)
  Call Extruder(128.40284)
  MoveL 6973 to (517.78, 555.37, 120) mm, rotated rx -180 ry 0 rz 160 deg; joints [12.592, 63.724, -10.386, -141.446, 59.797, 158.153]
  Call Extruder(133.49486)
  MoveL 6974 to (516.39, 555.8, 120) mm, rotated rx -180 ry 0 rz 160 deg; joints [12.678, 63.502, -9.936, -141.435, 60.007, 158.27]
  Set speed (16.1 mm/s)
  Call Extruder(136.79206)
  MoveL 6975 to (515.49, 556.06, 120) mm, rotated rx 180 ry 0 rz 160 deg; joints [12.732, 63.358, -9.643, -141.43, 60.143, 158.347]
  Set speed (16.1 mm/s)
  Call Extruder(140.25398)
  MoveL 6976 to (514.53, 556.31, 120) mm, rotated rx 180 ry 0 rz 160 deg; joints [12.787, 63.205, -9.334, -141.427, 60.286, 158.431]
  Set speed (16.1 mm/s)
  Call Extruder(144.80557)
  MoveL 6977 to (513.27, 556.62, 120) mm, rotated rx -180 ry 0 rz 160 deg; joints [12.858, 63.004, -8.926, -141.425, 60.473, 158.542]
  Set speed (16.1 mm/s)
  Call Extruder(153.33811)
  MoveL 6978 to (510.88, 557.13, 120) mm, rotated rx 180 ry 0 rz 160 deg; joints [12.982, 62.624, -8.156, -141.429, 60.824, 158.756]
  Set speed (16.1 mm/s)
  Call Extruder(161.71940)
  MoveL 6979 to (508.52, 557.53, 120) mm, rotated rx -180 ry 0 rz 160 deg; joints [13.094, 62.249, -7.393, -141.443, 61.167, 158.974]
  Set speed (16.1 mm/s)
  Call Extruder(169.83564)
  MoveL 6980 to (506.22, 557.82, 120) mm, rotated rx 180 ry 0 rz 160 deg; joints [13.193, 61.884, -6.65, -141.467, 61.498, 159.192]
  Set speed (16.1 mm/s)
  Call Extruder(178.33795)
  MoveL 6981 to (503.8, 558.03, 120) mm, rotated rx -180 ry 0 rz 160 deg; joints [13.286, 61.501, -5.869, -141.502, 61.843, 159.427]
  Set speed (16.1 mm/s)
  Call Extruder(186.71052)
  MoveL 6982 to (501.41, 558.14, 120) mm, rotated rx 180 ry 0 rz 160 deg; joints [13.367, 61.122, -5.097, -141.546, 62.179, 159.664]
  Call Extruder(194.93472)
  MoveL 6983 to (499.06, 558.15, 120) mm, rotated rx -180 ry 0 rz 160 deg; joints [13.436, 60.751, -4.338, -141.599, 62.506, 159.902]
  Set speed (10.0 mm/s)
  MoveL 6984 to (499.06, 558.15, 124) mm, rotated rx -180 ry 0 rz 160 deg; joints [13.436, 60.143, -4.112, -141.475, 62.207, 159.634]
  Set speed (120.0 mm/s)
  MoveL 6985 to (499.09, 556.18, 124) mm, rotated rx 180 ry 0 rz 160 deg; joints [13.197, 60.075, -3.973, -141.752, 62.18, 159.802]
  Set speed (16.2 mm/s)
  Call Extruder(202.74859)
  MoveL 6986 to (496.86, 556.1, 124) mm, rotated rx 180 ry 0 rz 160 deg; joints [13.25, 59.72, -3.252, -141.814, 62.486, 160.032]
  Set speed (16.2 mm/s)
  Call Extruder(211.07055)
  MoveL 6987 to (494.48, 555.91, 124) mm, rotated rx 180 ry 0 rz 160 deg; joints [13.297, 59.344, -2.485, -141.89, 62.809, 160.281]
  Call Extruder(219.01827)
  MoveL 6988 to (492.22, 555.65, 124) mm, rotated rx 180 ry 0 rz 160 deg; joints [13.329, 58.986, -1.755, -141.972, 63.113, 160.522]
  Call Extruder(227.00008)
  MoveL 6989 to (489.96, 555.28, 124) mm, rotated rx 180 ry 0 rz 160 deg; joints [13.35, 58.628, -1.025, -142.065, 63.413, 160.769]
  Call Extruder(235.15992)
  MoveL 6990 to (487.67, 554.82, 124) mm, rotated rx 180 ry 0 rz 160 deg; joints [13.36, 58.266, -0.284, -142.171, 63.716, 161.024]
  Set speed (16.2 mm/s)
  Call Extruder(239.11568)
  MoveL 6991 to (486.57, 554.55, 124) mm, rotated rx -180 ry 0 rz 160 deg; joints [13.36, 58.091, 0.073, -142.226, 63.86, 161.149]
  Call Extruder(243.12891)
  MoveL 6992 to (485.45, 554.27, 124) mm, rotated rx 180 ry 0 rz 160 deg; joints [13.358, 57.915, 0.434, -142.284, 64.005, 161.276]
  Set speed (16.2 mm/s)
  Call Extruder(251.01965)
  MoveL 6993 to (483.28, 553.64, 124) mm, rotated rx 180 ry 0 rz 160 deg; joints [13.343, 57.572, 1.139, -142.406, 64.286, 161.528]
  Set speed (16.2 mm/s)
  Call Extruder(258.94151)
  MoveL 6994 to (481.13, 552.92, 124) mm, rotated rx 180 ry 0 rz 160 deg; joints [13.317, 57.23, 1.839, -142.538, 64.563, 161.782]
  Set speed (16.2 mm/s)
  Call Extruder(263.19391)
  MoveL 6995 to (479.99, 552.5, 124) mm, rotated rx -180 ry 0 rz 160 deg; joints [13.298, 57.049, 2.212, -142.614, 64.709, 161.92]
  Set speed (16.2 mm/s)
  Call Extruder(267.13807)
  MoveL 6996 to (478.93, 552.09, 124) mm, rotated rx 180 ry 0 rz 160 deg; joints [13.277, 56.882, 2.555, -142.685, 64.843, 162.047]
  Set speed (16.2 mm/s)
  Call Extruder(274.12191)
  MoveL 6997 to (477.09, 551.31, 124) mm, rotated rx -180 ry 0 rz 160 deg; joints [13.233, 56.59, 3.156, -142.819, 65.076, 162.273]
  Set speed (16.2 mm/s)
  Call Extruder(279.16492)
  MoveL 6998 to (475.78, 550.7, 124) mm, rotated rx -180 ry 0 rz 160 deg; joints [13.195, 56.382, 3.586, -142.921, 65.24, 162.437]
  Set speed (16.2 mm/s)
  Call Extruder(285.19971)
  MoveL 6999 to (474.23, 549.94, 124) mm, rotated rx -180 ry 0 rz 160 deg; joints [13.144, 56.135, 4.094, -143.048, 65.434, 162.633]
  Set speed (16.1 mm/s)
  Call Extruder(291.24257)
  MoveL 7000 to (472.71, 549.12, 124) mm, rotated rx 180 ry 0 rz 160 deg; joints [13.084, 55.892, 4.596, -143.181, 65.623, 162.83]
  Set speed (16.2 mm/s)
  Call Extruder(294.57549)
  MoveL 7001 to (471.88, 548.64, 124) mm, rotated rx 180 ry 0 rz 160 deg; joints [13.048, 55.76, 4.87, -143.257, 65.726, 162.938]
  Set speed (16.2 mm/s)
  Call Extruder(298.44787)
  MoveL 7002 to (470.93, 548.08, 124) mm, rotated rx -180 ry 0 rz 160 deg; joints [13.003, 55.607, 5.186, -143.347, 65.844, 163.064]
  Set speed (16.2 mm/s)
  Call Extruder(303.22144)
  MoveL 7003 to (469.76, 547.36, 124) mm, rotated rx 180 ry 0 rz 160 deg; joints [12.944, 55.421, 5.571, -143.462, 65.986, 163.22]
  Call Extruder(307.29979)
  MoveL 7004 to (468.79, 546.72, 124) mm, rotated rx 180 ry 0 rz 160 deg; joints [12.89, 55.264, 5.896, -143.563, 66.106, 163.352]
  Set speed (16.2 mm/s)
  Call Extruder(311.23567)
  MoveL 7005 to (467.85, 546.08, 124) mm, rotated rx -180 ry 0 rz 160 deg; joints [12.835, 55.114, 6.206, -143.663, 66.219, 163.479]
  Set speed (16.2 mm/s)
  Call Extruder(315.17150)
  MoveL 7006 to (466.93, 545.43, 124) mm, rotated rx 180 ry 0 rz 160 deg; joints [12.777, 54.967, 6.513, -143.765, 66.331, 163.606]
  Set speed (16.2 mm/s)
  Call Extruder(319.29304)
  MoveL 7007 to (465.99, 544.72, 124) mm, rotated rx -180 ry 0 rz 160 deg; joints [12.712, 54.814, 6.829, -143.876, 66.445, 163.739]
  Set speed (16.2 mm/s)
  Call Extruder(323.19809)
  MoveL 7008 to (465.1, 544.04, 124) mm, rotated rx 180 ry 0 rz 160 deg; joints [12.648, 54.671, 7.126, -143.982, 66.552, 163.865]
  Set speed (16.2 mm/s)
  Call Extruder(326.58083)
  MoveL 7009 to (464.35, 543.43, 124) mm, rotated rx -180 ry 0 rz 160 deg; joints [12.591, 54.549, 7.38, -144.076, 66.642, 163.973]
  Set speed (16.1 mm/s)
  Call Extruder(332.37087)
  MoveL 7010 to (463.08, 542.36, 124) mm, rotated rx -180 ry 0 rz 160 deg; joints [12.487, 54.344, 7.807, -144.241, 66.793, 164.158]
  Set speed (16.2 mm/s)
  Call Extruder(335.30927)
  MoveL 7011 to (462.45, 541.8, 124) mm, rotated rx 180 ry 0 rz 160 deg; joints [12.431, 54.241, 8.02, -144.326, 66.868, 164.251]
  Set speed (16.2 mm/s)
  Call Extruder(339.27302)
  MoveL 7012 to (461.62, 541.03, 124) mm, rotated rx 180 ry 0 rz 160 deg; joints [12.353, 54.105, 8.304, -144.444, 66.967, 164.376]
  Set speed (16.2 mm/s)
  Call Extruder(343.27941)
  MoveL 7013 to (460.79, 540.24, 124) mm, rotated rx 180 ry 0 rz 160 deg; joints [12.272, 53.969, 8.587, -144.566, 67.065, 164.502]
  Call Extruder(347.33894)
  MoveL 7014 to (459.96, 539.42, 124) mm, rotated rx 180 ry 0 rz 160 deg; joints [12.186, 53.834, 8.869, -144.691, 67.162, 164.629]
  Call Extruder(351.37461)
  MoveL 7015 to (459.16, 538.59, 124) mm, rotated rx -180 ry 0 rz 160 deg; joints [12.098, 53.702, 9.144, -144.819, 67.256, 164.755]
  Set speed (16.2 mm/s)
  Call Extruder(355.33922)
  MoveL 7016 to (458.39, 537.75, 124) mm, rotated rx -180 ry 0 rz 160 deg; joints [12.008, 53.575, 9.411, -144.946, 67.346, 164.878]
  Set speed (16.2 mm/s)
  Call Extruder(359.33698)
  MoveL 7017 to (457.63, 536.9, 124) mm, rotated rx 180 ry 0 rz 160 deg; joints [11.914, 53.449, 9.674, -145.077, 67.434, 165.001]
  Set speed (16.2 mm/s)
  Call Extruder(362.90095)
  MoveL 7018 to (456.96, 536.12, 124) mm, rotated rx 180 ry 0 rz 160 deg; joints [11.828, 53.338, 9.905, -145.195, 67.511, 165.109]
  Set speed (16.2 mm/s)
  Call Extruder(367.47989)
  MoveL 7019 to (456.13, 535.11, 124) mm, rotated rx 180 ry 0 rz 160 deg; joints [11.715, 53.2, 10.195, -145.35, 67.606, 165.248]
  Set speed (16.2 mm/s)
  Call Extruder(371.39933)
  MoveL 7020 to (455.44, 534.22, 124) mm, rotated rx -180 ry 0 rz 160 deg; joints [11.614, 53.083, 10.438, -145.484, 67.685, 165.366]
  Set speed (16.2 mm/s)
  Call Extruder(375.43161)
  MoveL 7021 to (454.74, 533.3, 124) mm, rotated rx -180 ry 0 rz 160 deg; joints [11.508, 52.967, 10.682, -145.625, 67.763, 165.486]
  Call Extruder(379.42273)
  MoveL 7022 to (454.08, 532.37, 124) mm, rotated rx -180 ry 0 rz 160 deg; joints [11.399, 52.854, 10.919, -145.767, 67.839, 165.605]
  Call Extruder(383.44071)
  MoveL 7023 to (453.42, 531.42, 124) mm, rotated rx -180 ry 0 rz 160 deg; joints [11.288, 52.743, 11.152, -145.912, 67.912, 165.722]
  Call Extruder(387.45535)
  MoveL 7024 to (452.79, 530.46, 124) mm, rotated rx 180 ry 0 rz 160 deg; joints [11.173, 52.634, 11.379, -146.058, 67.982, 165.839]
  Set speed (16.2 mm/s)
  Call Extruder(391.44524)
  MoveL 7025 to (452.18, 529.49, 124) mm, rotated rx 180 ry 0 rz 160 deg; joints [11.057, 52.529, 11.6, -146.206, 68.05, 165.954]
  Set speed (16.2 mm/s)
  Call Extruder(395.45767)
  MoveL 7026 to (451.58, 528.51, 124) mm, rotated rx 180 ry 0 rz 160 deg; joints [10.938, 52.427, 11.815, -146.356, 68.115, 166.068]
  Set speed (16.2 mm/s)
  Call Extruder(399.46759)
  MoveL 7027 to (451.01, 527.51, 124) mm, rotated rx 180 ry 0 rz 160 deg; joints [10.815, 52.327, 12.025, -146.508, 68.177, 166.181]
  Call Extruder(403.46596)
  MoveL 7028 to (450.46, 526.51, 124) mm, rotated rx -180 ry 0 rz 160 deg; joints [10.691, 52.23, 12.228, -146.662, 68.237, 166.293]
  Set speed (16.2 mm/s)
  Call Extruder(407.48703)
  MoveL 7029 to (449.93, 525.49, 124) mm, rotated rx 180 ry 0 rz 160 deg; joints [10.563, 52.136, 12.426, -146.818, 68.293, 166.404]
  Set speed (16.2 mm/s)
  Call Extruder(411.58177)
  MoveL 7030 to (449.4, 524.44, 124) mm, rotated rx 180 ry 0 rz 160 deg; joints [10.431, 52.043, 12.622, -146.979, 68.348, 166.515]
  Call Extruder(419.40114)
  MoveL 7031 to (448.47, 522.4, 124) mm, rotated rx 180 ry 0 rz 160 deg; joints [10.171, 51.875, 12.977, -147.291, 68.445, 166.724]
  Set speed (16.2 mm/s)
  Call Extruder(423.63458)
  MoveL 7032 to (448, 521.28, 124) mm, rotated rx 180 ry 0 rz 160 deg; joints [10.026, 51.789, 13.158, -147.463, 68.492, 166.835]
  Set speed (16.2 mm/s)
  Call Extruder(427.41496)
  MoveL 7033 to (447.6, 520.28, 124) mm, rotated rx 180 ry 0 rz 160 deg; joints [9.895, 51.714, 13.316, -147.617, 68.533, 166.933]
  Set speed (16.2 mm/s)
  Call Extruder(431.66766)
  MoveL 7034 to (447.18, 519.14, 124) mm, rotated rx -180 ry 0 rz 160 deg; joints [9.746, 51.634, 13.485, -147.793, 68.574, 167.041]
  Call Extruder(435.60722)
  MoveL 7035 to (446.8, 518.07, 124) mm, rotated rx 180 ry 0 rz 160 deg; joints [9.606, 51.562, 13.637, -147.956, 68.61, 167.141]
  Call Extruder(439.68971)
  MoveL 7036 to (446.44, 516.96, 124) mm, rotated rx 180 ry 0 rz 160 deg; joints [9.458, 51.492, 13.784, -148.127, 68.644, 167.241]
  Set speed (16.1 mm/s)
  Call Extruder(443.57911)
  MoveL 7037 to (446.11, 515.9, 124) mm, rotated rx 180 ry 0 rz 160 deg; joints [9.315, 51.427, 13.921, -148.291, 68.674, 167.336]
  Call Extruder(447.72151)
  MoveL 7038 to (445.79, 514.76, 124) mm, rotated rx -180 ry 0 rz 160 deg; joints [9.161, 51.363, 14.058, -148.467, 68.701, 167.435]
  Set speed (16.2 mm/s)
  Call Extruder(451.55459)
  MoveL 7039 to (445.51, 513.7, 124) mm, rotated rx 180 ry 0 rz 160 deg; joints [9.018, 51.305, 14.18, -148.63, 68.725, 167.526]
  Set speed (16.1 mm/s)
  Call Extruder(455.08215)
  MoveL 7040 to (445.27, 512.72, 124) mm, rotated rx 180 ry 0 rz 160 deg; joints [8.884, 51.255, 14.285, -148.782, 68.744, 167.608]
  Set speed (16.1 mm/s)
  Call Extruder(459.60503)
  MoveL 7041 to (444.99, 511.45, 124) mm, rotated rx 180 ry 0 rz 160 deg; joints [8.711, 51.194, 14.414, -148.977, 68.765, 167.711]
  Set speed (16.2 mm/s)
  Call Extruder(467.82058)
  MoveL 7042 to (444.56, 509.14, 124) mm, rotated rx 180 ry 0 rz 160 deg; joints [8.391, 51.095, 14.624, -149.334, 68.792, 167.894]
  Set speed (16.2 mm/s)
  Call Extruder(475.84535)
  MoveL 7043 to (444.24, 506.86, 124) mm, rotated rx -180 ry 0 rz 160 deg; joints [8.073, 51.012, 14.801, -149.686, 68.807, 168.065]
  Set speed (16.2 mm/s)
  Call Extruder(483.86382)
  MoveL 7044 to (444, 504.58, 124) mm, rotated rx -180 ry 0 rz 160 deg; joints [7.752, 50.941, 14.95, -150.039, 68.809, 168.229]
  Call Extruder(491.69044)
  MoveL 7045 to (443.86, 502.34, 124) mm, rotated rx 180 ry 0 rz 160 deg; joints [7.434, 50.886, 15.067, -150.385, 68.798, 168.383]
  Set speed (16.2 mm/s)
  Call Extruder(499.80493)
  MoveL 7046 to (443.81, 500.01, 124) mm, rotated rx -180 ry 0 rz 160 deg; joints [7.101, 50.842, 15.16, -150.744, 68.774, 168.535]
  Set speed (16.2 mm/s)
  Call Extruder(507.12206)
  MoveL 7047 to (443.85, 497.92, 124) mm, rotated rx 180 ry 0 rz 160 deg; joints [6.799, 50.815, 15.218, -151.067, 68.741, 168.667]
  Set speed (16.2 mm/s)
  Call Extruder(514.24372)
  MoveL 7048 to (443.96, 495.88, 124) mm, rotated rx -180 ry 0 rz 160 deg; joints [6.505, 50.799, 15.253, -151.381, 68.7, 168.789]
  Call Extruder(521.36753)
  MoveL 7049 to (444.15, 493.85, 124) mm, rotated rx 180 ry 0 rz 160 deg; joints [6.209, 50.794, 15.263, -151.693, 68.648, 168.905]
  Set speed (16.2 mm/s)
  Call Extruder(528.67979)
  MoveL 7050 to (444.42, 491.77, 124) mm, rotated rx -180 ry 0 rz 160 deg; joints [5.906, 50.8, 15.251, -152.011, 68.583, 169.018]
  Set speed (16.2 mm/s)
  Call Extruder(535.71236)
  MoveL 7051 to (444.75, 489.78, 124) mm, rotated rx 180 ry 0 rz 160 deg; joints [5.615, 50.816, 15.215, -152.315, 68.512, 169.121]
  Set speed (16.2 mm/s)
  Call Extruder(543.10448)
  MoveL 7052 to (445.18, 487.7, 124) mm, rotated rx 180 ry 0 rz 160 deg; joints [5.31, 50.845, 15.154, -152.631, 68.426, 169.223]
  Set speed (16.2 mm/s)
  Call Extruder(550.25284)
  MoveL 7053 to (445.66, 485.72, 124) mm, rotated rx 180 ry 0 rz 160 deg; joints [5.017, 50.884, 15.071, -152.932, 68.332, 169.315]
  Set speed (16.2 mm/s)
  Call Extruder(557.54745)
  MoveL 7054 to (446.23, 483.7, 124) mm, rotated rx 180 ry 0 rz 160 deg; joints [4.721, 50.935, 14.964, -153.236, 68.227, 169.404]
  Set speed (16.2 mm/s)
  Call Extruder(564.75886)
  MoveL 7055 to (446.86, 481.74, 124) mm, rotated rx 180 ry 0 rz 160 deg; joints [4.431, 50.996, 14.835, -153.531, 68.113, 169.485]
  Set speed (16.2 mm/s)
  Call Extruder(572.09248)
  MoveL 7056 to (447.59, 479.76, 124) mm, rotated rx -180 ry 0 rz 160 deg; joints [4.139, 51.069, 14.679, -153.825, 67.986, 169.561]
  Set speed (16.2 mm/s)
  Call Extruder(579.31343)
  MoveL 7057 to (448.36, 477.85, 124) mm, rotated rx 180 ry 0 rz 160 deg; joints [3.857, 51.152, 14.503, -154.108, 67.852, 169.63]
  Set speed (16.2 mm/s)
  Call Extruder(586.52203)
  MoveL 7058 to (449.21, 475.97, 124) mm, rotated rx -180 ry 0 rz 160 deg; joints [3.579, 51.246, 14.305, -154.385, 67.708, 169.693]
  Set speed (16.2 mm/s)
  Call Extruder(593.65889)
  MoveL 7059 to (450.12, 474.14, 124) mm, rotated rx -180 ry 0 rz 160 deg; joints [3.309, 51.349, 14.087, -154.652, 67.556, 169.748]
  Set speed (16.2 mm/s)
  Call Extruder(600.87426)
  MoveL 7060 to (451.11, 472.32, 124) mm, rotated rx -180 ry 0 rz 160 deg; joints [3.042, 51.463, 13.845, -154.914, 67.393, 169.799]
  Set speed (16.2 mm/s)
  Call Extruder(608.13405)
  MoveL 7061 to (452.16, 470.53, 124) mm, rotated rx -180 ry 0 rz 160 deg; joints [2.779, 51.589, 13.58, -155.17, 67.22, 169.843]
  Set speed (16.2 mm/s)
  Call Extruder(615.30930)
  MoveL 7062 to (453.27, 468.8, 124) mm, rotated rx -180 ry 0 rz 160 deg; joints [2.525, 51.723, 13.296, -155.414, 67.04, 169.881]
  Set speed (16.2 mm/s)
  Call Extruder(622.53085)
  MoveL 7063 to (454.45, 467.1, 124) mm, rotated rx -180 ry 0 rz 160 deg; joints [2.277, 51.869, 12.99, -155.652, 66.85, 169.912]
  Set speed (16.2 mm/s)
  Call Extruder(629.84455)
  MoveL 7064 to (455.71, 465.42, 124) mm, rotated rx -180 ry 0 rz 160 deg; joints [2.033, 52.026, 12.659, -155.882, 66.648, 169.937]
  Call Extruder(636.86304)
  MoveL 7065 to (456.98, 463.86, 124) mm, rotated rx -180 ry 0 rz 160 deg; joints [1.807, 52.186, 12.322, -156.094, 66.447, 169.956]
  Set speed (16.2 mm/s)
  Call Extruder(644.04649)
  MoveL 7066 to (458.33, 462.31, 124) mm, rotated rx 180 ry 0 rz 160 deg; joints [1.583, 52.359, 11.958, -156.301, 66.234, 169.968]
  Set speed (16.2 mm/s)
  Call Extruder(651.49908)
  MoveL 7067 to (459.8, 460.75, 124) mm, rotated rx 180 ry 0 rz 160 deg; joints [1.36, 52.548, 11.56, -156.504, 66.004, 169.974]
  Set speed (16.2 mm/s)
  Call Extruder(658.47929)
  MoveL 7068 to (461.22, 459.34, 124) mm, rotated rx 180 ry 0 rz 160 deg; joints [1.158, 52.734, 11.17, -156.685, 65.781, 169.974]
  Set speed (16.2 mm/s)
  Call Extruder(665.84266)
  MoveL 7069 to (462.77, 457.92, 124) mm, rotated rx 180 ry 0 rz 160 deg; joints [0.956, 52.939, 10.739, -156.864, 65.539, 169.967]
  Call Extruder(673.14817)
  MoveL 7070 to (464.37, 456.56, 124) mm, rotated rx -180 ry 0 rz 160 deg; joints [0.764, 53.152, 10.294, -157.03, 65.292, 169.953]
  Set speed (16.2 mm/s)
  Call Extruder(680.20864)
  MoveL 7071 to (465.95, 455.31, 124) mm, rotated rx 180 ry 0 rz 160 deg; joints [0.588, 53.365, 9.848, -157.179, 65.046, 169.933]
  Set speed (16.2 mm/s)
  Call Extruder(686.99149)
  MoveL 7072 to (467.52, 454.15, 124) mm, rotated rx -180 ry 0 rz 160 deg; joints [0.428, 53.578, 9.404, -157.311, 64.805, 169.908]
  Set speed (16.2 mm/s)
  Call Extruder(694.77103)
  MoveL 7073 to (469.36, 452.9, 124) mm, rotated rx -180 ry 0 rz 160 deg; joints [0.255, 53.83, 8.878, -157.45, 64.521, 169.872]
  Set speed (16.2 mm/s)
  Call Extruder(702.04307)
  MoveL 7074 to (471.13, 451.8, 124) mm, rotated rx 180 ry 0 rz 160 deg; joints [0.103, 54.073, 8.37, -157.567, 64.25, 169.832]
  Set speed (16.2 mm/s)
  Call Extruder(709.24056)
  MoveL 7075 to (472.92, 450.77, 124) mm, rotated rx -180 ry 0 rz 160 deg; joints [-0.037, 54.322, 7.852, -157.67, 63.977, 169.785]
  Call Extruder(716.42163)
  MoveL 7076 to (474.74, 449.81, 124) mm, rotated rx 180 ry 0 rz 160 deg; joints [-0.166, 54.577, 7.322, -157.761, 63.699, 169.731]
  Set speed (16.2 mm/s)
  Call Extruder(723.64601)
  MoveL 7077 to (476.6, 448.92, 124) mm, rotated rx 180 ry 0 rz 160 deg; joints [-0.286, 54.84, 6.775, -157.839, 63.415, 169.67]
  Set speed (16.2 mm/s)
  Call Extruder(730.92162)
  MoveL 7078 to (478.51, 448.08, 124) mm, rotated rx 180 ry 0 rz 160 deg; joints [-0.397, 55.112, 6.212, -157.906, 63.125, 169.602]
  Set speed (16.2 mm/s)
  Call Extruder(738.02335)
  MoveL 7079 to (480.41, 447.34, 124) mm, rotated rx 180 ry 0 rz 160 deg; joints [-0.494, 55.383, 5.65, -157.957, 62.838, 169.528]
  Set speed (16.2 mm/s)
  Call Extruder(745.28293)
  MoveL 7080 to (482.37, 446.65, 124) mm, rotated rx 180 ry 0 rz 160 deg; joints [-0.583, 55.666, 5.064, -157.997, 62.541, 169.445]
  Set speed (16.2 mm/s)
  Call Extruder(752.50876)
  MoveL 7081 to (484.35, 446.04, 124) mm, rotated rx -180 ry 0 rz 160 deg; joints [-0.662, 55.953, 4.47, -158.024, 62.242, 169.356]
  Set speed (16.2 mm/s)
  Call Extruder(759.88887)
  MoveL 7082 to (486.39, 445.49, 124) mm, rotated rx 180 ry 0 rz 160 deg; joints [-0.731, 56.252, 3.853, -158.039, 61.934, 169.258]
  Set speed (16.2 mm/s)
  Call Extruder(766.99438)
  MoveL 7083 to (488.38, 445.03, 124) mm, rotated rx -180 ry 0 rz 160 deg; joints [-0.787, 56.545, 3.25, -158.039, 61.635, 169.155]
  Set speed (16.2 mm/s)
  Call Extruder(774.04442)
  MoveL 7084 to (490.36, 444.65, 124) mm, rotated rx -180 ry 0 rz 160 deg; joints [-0.833, 56.84, 2.643, -158.027, 61.337, 169.047]
  Set speed (16.2 mm/s)
  Call Extruder(781.00031)
  MoveL 7085 to (492.33, 444.34, 124) mm, rotated rx 180 ry 0 rz 160 deg; joints [-0.87, 57.134, 2.037, -158.004, 61.042, 168.934]
  Call Extruder(788.60021)
  MoveL 7086 to (494.49, 444.09, 124) mm, rotated rx -180 ry 0 rz 160 deg; joints [-0.898, 57.46, 1.367, -157.964, 60.718, 168.802]
  Set speed (16.2 mm/s)
  Call Extruder(795.68553)
  MoveL 7087 to (496.52, 443.92, 124) mm, rotated rx 180 ry 0 rz 160 deg; joints [-0.915, 57.768, 0.737, -157.914, 60.415, 168.672]
  Set speed (16.2 mm/s)
  Call Extruder(803.09224)
  MoveL 7088 to (498.64, 443.83, 124) mm, rotated rx 180 ry 0 rz 160 deg; joints [-0.923, 58.092, 0.071, -157.85, 60.098, 168.528]
  Set speed (16.2 mm/s)
  Call Extruder(810.22205)
  MoveL 7089 to (500.68, 443.82, 124) mm, rotated rx 180 ry 0 rz 160 deg; joints [-0.92, 58.408, -0.574, -157.774, 59.793, 168.383]
  Set speed (16.2 mm/s)
  Call Extruder(817.51298)
  MoveL 7090 to (502.77, 443.88, 124) mm, rotated rx 180 ry 0 rz 160 deg; joints [-0.908, 58.733, -1.239, -157.685, 59.481, 168.226]
  Call Extruder(824.63893)
  MoveL 7091 to (504.81, 444.02, 124) mm, rotated rx -180 ry 0 rz 160 deg; joints [-0.886, 59.053, -1.892, -157.586, 59.177, 168.067]
  Set speed (16.2 mm/s)
  Call Extruder(831.67742)
  MoveL 7092 to (506.82, 444.23, 124) mm, rotated rx -180 ry 0 rz 160 deg; joints [-0.856, 59.37, -2.539, -157.475, 58.879, 167.902]
  Set speed (16.2 mm/s)
  Call Extruder(839.09787)
  MoveL 7093 to (508.92, 444.53, 124) mm, rotated rx -180 ry 0 rz 160 deg; joints [-0.815, 59.706, -3.223, -157.347, 58.566, 167.721]
  Set speed (16.2 mm/s)
  Call Extruder(846.37014)
  MoveL 7094 to (510.97, 444.89, 124) mm, rotated rx -180 ry 0 rz 160 deg; joints [-0.765, 60.036, -3.894, -157.209, 58.262, 167.537]
  Set speed (16.2 mm/s)
  Call Extruder(853.35101)
  MoveL 7095 to (512.93, 445.32, 124) mm, rotated rx 180 ry 0 rz 160 deg; joints [-0.709, 60.353, -4.538, -157.066, 57.973, 167.353]
  Set speed (16.2 mm/s)
  Call Extruder(860.72139)
  MoveL 7096 to (514.98, 445.85, 124) mm, rotated rx 180 ry 0 rz 160 deg; joints [-0.641, 60.688, -5.218, -156.903, 57.67, 167.152]
  Call Extruder(867.93932)
  MoveL 7097 to (516.96, 446.43, 124) mm, rotated rx -180 ry 0 rz 160 deg; joints [-0.566, 61.016, -5.883, -156.732, 57.377, 166.948]
  Set speed (16.2 mm/s)
  Call Extruder(875.24854)
  MoveL 7098 to (518.94, 447.11, 124) mm, rotated rx -180 ry 0 rz 160 deg; joints [-0.482, 61.346, -6.553, -156.547, 57.085, 166.735]
  Set speed (16.2 mm/s)
  Call Extruder(882.36198)
  MoveL 7099 to (520.85, 447.82, 124) mm, rotated rx -180 ry 0 rz 160 deg; joints [-0.392, 61.668, -7.203, -156.358, 56.804, 166.522]
  Call Extruder(889.66452)
  MoveL 7100 to (522.78, 448.64, 124) mm, rotated rx 180 ry 0 rz 160 deg; joints [-0.292, 61.995, -7.865, -156.152, 56.522, 166.296]
  Set speed (16.2 mm/s)
  Call Extruder(896.64056)
  MoveL 7101 to (524.59, 449.48, 124) mm, rotated rx -180 ry 0 rz 160 deg; joints [-0.189, 62.307, -8.494, -155.946, 56.256, 166.075]
  Call Extruder(903.89319)
  MoveL 7102 to (526.45, 450.43, 124) mm, rotated rx 180 ry 0 rz 160 deg; joints [-0.074, 62.628, -9.142, -155.723, 55.986, 165.839]
  Set speed (16.2 mm/s)
  Call Extruder(911.31483)
  MoveL 7103 to (528.3, 451.46, 124) mm, rotated rx -180 ry 0 rz 160 deg; joints [0.05, 62.954, -9.798, -155.484, 55.715, 165.592]
  Call Extruder(918.43060)
  MoveL 7104 to (530.05, 452.52, 124) mm, rotated rx -180 ry 0 rz 160 deg; joints [0.177, 63.263, -10.42, -155.246, 55.463, 165.35]
  Set speed (16.2 mm/s)
  Call Extruder(925.74898)
  MoveL 7105 to (531.8, 453.68, 124) mm, rotated rx -180 ry 0 rz 160 deg; joints [0.314, 63.576, -11.051, -154.993, 55.21, 165.097]
  Call Extruder(932.87143)
  MoveL 7106 to (533.46, 454.86, 124) mm, rotated rx 180 ry 0 rz 160 deg; joints [0.454, 63.877, -11.655, -154.739, 54.971, 164.845]
  Call Extruder(940.13684)
  MoveL 7107 to (535.11, 456.13, 124) mm, rotated rx -180 ry 0 rz 160 deg; joints [0.602, 64.179, -12.262, -154.471, 54.735, 164.584]
  Call Extruder(947.30790)
  MoveL 7108 to (536.69, 457.45, 124) mm, rotated rx -180 ry 0 rz 160 deg; joints [0.755, 64.472, -12.85, -154.2, 54.51, 164.323]
  Set speed (16.2 mm/s)
  Call Extruder(954.61364)
  MoveL 7109 to (538.25, 458.84, 124) mm, rotated rx 180 ry 0 rz 160 deg; joints [0.917, 64.765, -13.437, -153.917, 54.29, 164.054]
  Set speed (16.2 mm/s)
  Call Extruder(961.95042)
  MoveL 7110 to (539.76, 460.3, 124) mm, rotated rx -180 ry 0 rz 160 deg; joints [1.085, 65.053, -14.014, -153.626, 54.078, 163.78]
  Set speed (16.2 mm/s)
  Call Extruder(966.59183)
  MoveL 7111 to (540.69, 461.26, 124) mm, rotated rx -180 ry 0 rz 160 deg; joints [1.194, 65.232, -14.371, -153.438, 53.948, 163.605]
  Set speed (16.2 mm/s)
  Call Extruder(969.79596)
  MoveL 7112 to (541.32, 461.93, 124) mm, rotated rx -180 ry 0 rz 160 deg; joints [1.271, 65.353, -14.614, -153.307, 53.862, 163.484]
  Set speed (16.2 mm/s)
  Call Extruder(973.80876)
  MoveL 7113 to (542.09, 462.78, 124) mm, rotated rx -180 ry 0 rz 160 deg; joints [1.368, 65.503, -14.914, -153.142, 53.755, 163.332]
  Call Extruder(977.72522)
  MoveL 7114 to (542.83, 463.63, 124) mm, rotated rx -180 ry 0 rz 160 deg; joints [1.465, 65.647, -15.203, -152.979, 53.655, 163.183]
  Set speed (16.2 mm/s)
  Call Extruder(981.77159)
  MoveL 7115 to (543.57, 464.52, 124) mm, rotated rx -180 ry 0 rz 160 deg; joints [1.566, 65.794, -15.496, -152.809, 53.554, 163.028]
  Set speed (16.2 mm/s)
  Call Extruder(985.68850)
  MoveL 7116 to (544.27, 465.4, 124) mm, rotated rx 180 ry 0 rz 160 deg; joints [1.666, 65.934, -15.775, -152.644, 53.459, 162.879]
  Call Extruder(989.71259)
  MoveL 7117 to (544.97, 466.31, 124) mm, rotated rx -180 ry 0 rz 160 deg; joints [1.77, 66.075, -16.056, -152.472, 53.365, 162.724]
  Set speed (16.2 mm/s)
  Call Extruder(993.79262)
  MoveL 7118 to (545.66, 467.26, 124) mm, rotated rx -180 ry 0 rz 160 deg; joints [1.876, 66.215, -16.337, -152.297, 53.273, 162.568]
  Set speed (16.2 mm/s)
  Call Extruder(997.74963)
  MoveL 7119 to (546.31, 468.19, 124) mm, rotated rx -180 ry 0 rz 160 deg; joints [1.981, 66.348, -16.602, -152.126, 53.187, 162.416]
  Set speed (16.2 mm/s)
  Call Extruder(1001.76206)
  MoveL 7120 to (546.95, 469.14, 124) mm, rotated rx 180 ry 0 rz 160 deg; joints [2.088, 66.481, -16.866, -151.952, 53.103, 162.262]
  Set speed (16.2 mm/s)
  Call Extruder(1005.75922)
  MoveL 7121 to (547.57, 470.1, 124) mm, rotated rx -180 ry 0 rz 160 deg; joints [2.197, 66.61, -17.124, -151.777, 53.023, 162.109]
  Set speed (16.2 mm/s)
  Call Extruder(1009.78065)
  MoveL 7122 to (548.17, 471.09, 124) mm, rotated rx 180 ry 0 rz 160 deg; joints [2.307, 66.737, -17.376, -151.601, 52.947, 161.955]
  Set speed (16.2 mm/s)
  Call Extruder(1013.87471)
  MoveL 7123 to (548.77, 472.1, 124) mm, rotated rx -180 ry 0 rz 160 deg; joints [2.421, 66.862, -17.627, -151.421, 52.872, 161.799]
  Set speed (16.2 mm/s)
  Call Extruder(1020.00664)
  MoveL 7124 to (549.62, 473.63, 124) mm, rotated rx 180 ry 0 rz 160 deg; joints [2.593, 67.046, -17.992, -151.15, 52.767, 161.565]
  Set speed (16.2 mm/s)
  Call Extruder(1025.05957)
  MoveL 7125 to (550.28, 474.92, 124) mm, rotated rx -180 ry 0 rz 160 deg; joints [2.737, 67.19, -18.279, -150.925, 52.687, 161.374]
  Set speed (16.2 mm/s)
  Call Extruder(1029.81072)
  MoveL 7126 to (550.87, 476.15, 124) mm, rotated rx 180 ry 0 rz 160 deg; joints [2.873, 67.322, -18.542, -150.714, 52.617, 161.195]
  Call Extruder(1034.12116)
  MoveL 7127 to (551.39, 477.27, 124) mm, rotated rx -180 ry 0 rz 160 deg; joints [2.999, 67.437, -18.772, -150.522, 52.558, 161.034]
  Set speed (16.2 mm/s)
  Call Extruder(1041.50703)
  MoveL 7128 to (552.2, 479.22, 124) mm, rotated rx -180 ry 0 rz 160 deg; joints [3.216, 67.625, -19.146, -150.192, 52.468, 160.761]
  Set speed (16.1 mm/s)
  Call Extruder(1045.97889)
  MoveL 7129 to (552.66, 480.42, 124) mm, rotated rx -180 ry 0 rz 160 deg; joints [3.349, 67.732, -19.358, -149.993, 52.42, 160.598]
  Set speed (16.2 mm/s)
  Call Extruder(1049.94393)
  MoveL 7130 to (553.05, 481.48, 124) mm, rotated rx -180 ry 0 rz 160 deg; joints [3.468, 67.825, -19.543, -149.817, 52.38, 160.453]
  Set speed (16.2 mm/s)
  Call Extruder(1054.01740)
  MoveL 7131 to (553.42, 482.59, 124) mm, rotated rx -180 ry 0 rz 160 deg; joints [3.591, 67.915, -19.721, -149.636, 52.345, 160.308]
  Call Extruder(1058.21608)
  MoveL 7132 to (553.78, 483.73, 124) mm, rotated rx -180 ry 0 rz 160 deg; joints [3.718, 68.005, -19.901, -149.45, 52.311, 160.158]
  Set speed (16.2 mm/s)
  Call Extruder(1062.04262)
  MoveL 7133 to (554.08, 484.79, 124) mm, rotated rx -180 ry 0 rz 160 deg; joints [3.835, 68.082, -20.054, -149.281, 52.286, 160.024]
  Set speed (16.2 mm/s)
  Call Extruder(1065.84655)
  MoveL 7134 to (554.37, 485.84, 124) mm, rotated rx 180 ry 0 rz 160 deg; joints [3.952, 68.157, -20.202, -149.113, 52.263, 159.892]
  Set speed (16.2 mm/s)
  Call Extruder(1070.07585)
  MoveL 7135 to (554.66, 487.01, 124) mm, rotated rx 180 ry 0 rz 160 deg; joints [4.083, 68.234, -20.355, -148.927, 52.243, 159.747]
  Call Extruder(1074.06678)
  MoveL 7136 to (554.92, 488.13, 124) mm, rotated rx 180 ry 0 rz 160 deg; joints [4.206, 68.304, -20.495, -148.753, 52.226, 159.612]
  Set speed (16.2 mm/s)
  Call Extruder(1082.08578)
  MoveL 7137 to (555.36, 490.38, 124) mm, rotated rx -180 ry 0 rz 160 deg; joints [4.457, 68.432, -20.749, -148.404, 52.207, 159.347]
  Set speed (16.2 mm/s)
  Call Extruder(1090.10099)
  MoveL 7138 to (555.7, 492.65, 124) mm, rotated rx 180 ry 0 rz 160 deg; joints [4.71, 68.543, -20.968, -148.061, 52.204, 159.091]
  Set speed (16.2 mm/s)
  Call Extruder(1098.22154)
  MoveL 7139 to (555.96, 494.96, 124) mm, rotated rx -180 ry 0 rz 160 deg; joints [4.968, 68.638, -21.158, -147.717, 52.217, 158.841]
  Set speed (16.2 mm/s)
  Call Extruder(1106.13963)
  MoveL 7140 to (556.12, 497.23, 124) mm, rotated rx 180 ry 0 rz 160 deg; joints [5.221, 68.714, -21.308, -147.388, 52.246, 158.607]
  Call Extruder(1114.16782)
  MoveL 7141 to (556.19, 499.53, 124) mm, rotated rx -180 ry 0 rz 160 deg; joints [5.479, 68.774, -21.427, -147.06, 52.291, 158.381]
  Set speed (16.2 mm/s)
  Call Extruder(1122.03057)
  MoveL 7142 to (556.16, 501.78, 124) mm, rotated rx -180 ry 0 rz 160 deg; joints [5.733, 68.815, -21.508, -146.745, 52.351, 158.172]
  Set speed (16.2 mm/s)
  Call Extruder(1130.18603)
  MoveL 7143 to (556.04, 504.12, 124) mm, rotated rx 180 ry 0 rz 160 deg; joints [5.996, 68.84, -21.557, -146.427, 52.429, 157.967]
  Call Extruder(1138.10379)
  MoveL 7144 to (555.82, 506.38, 124) mm, rotated rx 180 ry 0 rz 160 deg; joints [6.252, 68.846, -21.569, -146.125, 52.52, 157.78]
  Set speed (16.2 mm/s)
  Call Extruder(1146.32920)
  MoveL 7145 to (555.51, 508.71, 124) mm, rotated rx 180 ry 0 rz 160 deg; joints [6.518, 68.835, -21.547, -145.82, 52.63, 157.6]
  Set speed (16.2 mm/s)
  Call Extruder(1154.32719)
  MoveL 7146 to (555.1, 510.97, 124) mm, rotated rx -180 ry 0 rz 160 deg; joints [6.776, 68.805, -21.488, -145.533, 52.753, 157.439]
  Set speed (16.2 mm/s)
  Call Extruder(1162.64222)
  MoveL 7147 to (554.59, 513.3, 124) mm, rotated rx -180 ry 0 rz 160 deg; joints [7.043, 68.757, -21.392, -145.244, 52.895, 157.286]
  Set speed (16.2 mm/s)
  Call Extruder(1170.46162)
  MoveL 7148 to (554.02, 515.46, 124) mm, rotated rx 180 ry 0 rz 160 deg; joints [7.294, 68.693, -21.266, -144.981, 53.044, 157.156]
  Set speed (16.2 mm/s)
  Call Extruder(1178.11905)
  MoveL 7149 to (553.37, 517.56, 124) mm, rotated rx -180 ry 0 rz 160 deg; joints [7.539, 68.614, -21.11, -144.733, 53.202, 157.043]
  Set speed (16.2 mm/s)
  Call Extruder(1182.33677)
  MoveL 7150 to (552.98, 518.7, 124) mm, rotated rx -180 ry 0 rz 160 deg; joints [7.672, 68.563, -21.009, -144.601, 53.295, 156.987]
  Set speed (16.2 mm/s)
  Call Extruder(1186.29935)
  MoveL 7151 to (552.59, 519.77, 124) mm, rotated rx 180 ry 0 rz 160 deg; joints [7.798, 68.514, -20.91, -144.478, 53.384, 156.936]
  Set speed (16.2 mm/s)
  Call Extruder(1194.36873)
  MoveL 7152 to (551.74, 521.92, 124) mm, rotated rx -180 ry 0 rz 160 deg; joints [8.052, 68.398, -20.681, -144.236, 53.576, 156.846]
  Call Extruder(1202.31552)
  MoveL 7153 to (550.8, 524, 124) mm, rotated rx -180 ry 0 rz 160 deg; joints [8.3, 68.267, -20.42, -144.009, 53.779, 156.772]
  Set speed (16.2 mm/s)
  Call Extruder(1204.46317)
  MoveL 7154 to (550.53, 524.55, 124) mm, rotated rx -180 ry 0 rz 160 deg; joints [8.367, 68.227, -20.341, -143.95, 53.837, 156.756]
  Set speed (16.2 mm/s)
  Call Extruder(1205.45342)
  MoveL 7155 to (550.41, 524.81, 124) mm, rotated rx -180 ry 0 rz 160 deg; joints [8.398, 68.211, -20.309, -143.922, 53.862, 156.747]
  Call Extruder(1210.51577)
  MoveL 7156 to (549.76, 526.1, 124) mm, rotated rx 180 ry 0 rz 160 deg; joints [8.554, 68.115, -20.119, -143.785, 54, 156.711]
  Set speed (16.2 mm/s)
  Call Extruder(1213.60473)
  MoveL 7157 to (549.34, 526.88, 124) mm, rotated rx 180 ry 0 rz 160 deg; joints [8.648, 68.053, -19.996, -143.704, 54.087, 156.693]
  Call Extruder(1218.27064)
  MoveL 7158 to (548.68, 528.05, 124) mm, rotated rx -180 ry 0 rz 160 deg; joints [8.791, 67.956, -19.803, -143.583, 54.22, 156.668]
  Set speed (16.2 mm/s)
  Call Extruder(1223.32825)
  MoveL 7159 to (547.94, 529.3, 124) mm, rotated rx 180 ry 0 rz 160 deg; joints [8.944, 67.845, -19.582, -143.457, 54.369, 156.648]
  Set speed (16.2 mm/s)
  Call Extruder(1226.31214)
  MoveL 7160 to (547.49, 530.02, 124) mm, rotated rx 180 ry 0 rz 160 deg; joints [9.034, 67.777, -19.446, -143.385, 54.459, 156.638]
  Set speed (16.2 mm/s)
  Call Extruder(1230.36648)
  MoveL 7161 to (546.86, 531, 124) mm, rotated rx -180 ry 0 rz 160 deg; joints [9.155, 67.68, -19.255, -143.289, 54.583, 156.629]
  Call Extruder(1234.34601)
  MoveL 7162 to (546.22, 531.94, 124) mm, rotated rx 180 ry 0 rz 160 deg; joints [9.273, 67.583, -19.061, -143.197, 54.707, 156.623]
  Set speed (16.2 mm/s)
  Call Extruder(1238.47398)
  MoveL 7163 to (545.54, 532.91, 124) mm, rotated rx 180 ry 0 rz 160 deg; joints [9.394, 67.477, -18.85, -143.105, 54.839, 156.621]
  Set speed (16.2 mm/s)
  Call Extruder(1242.50932)
  MoveL 7164 to (544.85, 533.84, 124) mm, rotated rx 180 ry 0 rz 160 deg; joints [9.512, 67.371, -18.639, -143.017, 54.97, 156.622]
  Set speed (16.2 mm/s)
  Call Extruder(1246.36116)
  MoveL 7165 to (544.18, 534.71, 124) mm, rotated rx -180 ry 0 rz 160 deg; joints [9.624, 67.266, -18.431, -142.935, 55.097, 156.627]
  Call Extruder(1250.41175)
  MoveL 7166 to (543.45, 535.62, 124) mm, rotated rx 180 ry 0 rz 160 deg; joints [9.74, 67.152, -18.204, -142.853, 55.233, 156.635]
  Set speed (16.2 mm/s)
  Call Extruder(1254.45266)
  MoveL 7167 to (542.71, 536.51, 124) mm, rotated rx 180 ry 0 rz 160 deg; joints [9.855, 67.035, -17.972, -142.773, 55.371, 156.647]
  Set speed (16.2 mm/s)
  Call Extruder(1258.42905)
  MoveL 7168 to (541.96, 537.37, 124) mm, rotated rx -180 ry 0 rz 160 deg; joints [9.967, 66.918, -17.737, -142.697, 55.508, 156.662]
  Set speed (16.2 mm/s)
  Call Extruder(1262.49683)
  MoveL 7169 to (541.18, 538.23, 124) mm, rotated rx 180 ry 0 rz 160 deg; joints [10.08, 66.794, -17.49, -142.622, 55.651, 156.682]
  Set speed (16.2 mm/s)
  Call Extruder(1266.42635)
  MoveL 7170 to (540.4, 539.05, 124) mm, rotated rx 180 ry 0 rz 160 deg; joints [10.188, 66.671, -17.246, -142.552, 55.79, 156.703]
  Set speed (16.2 mm/s)
  Call Extruder(1270.48874)
  MoveL 7171 to (539.59, 539.88, 124) mm, rotated rx 180 ry 0 rz 160 deg; joints [10.299, 66.541, -16.988, -142.482, 55.936, 156.729]
  Set speed (16.2 mm/s)
  Call Extruder(1274.50188)
  MoveL 7172 to (538.76, 540.68, 124) mm, rotated rx 180 ry 0 rz 160 deg; joints [10.407, 66.41, -16.725, -142.416, 56.082, 156.758]
  Call Extruder(1278.57132)
  MoveL 7173 to (537.91, 541.47, 124) mm, rotated rx -180 ry 0 rz 160 deg; joints [10.515, 66.274, -16.454, -142.352, 56.232, 156.791]
  Set speed (16.2 mm/s)
  Call Extruder(1282.60362)
  MoveL 7174 to (537.05, 542.24, 124) mm, rotated rx 180 ry 0 rz 160 deg; joints [10.621, 66.137, -16.181, -142.29, 56.382, 156.826]
  Set speed (16.2 mm/s)
  Call Extruder(1286.56005)
  MoveL 7175 to (536.19, 542.98, 124) mm, rotated rx -180 ry 0 rz 160 deg; joints [10.724, 66, -15.906, -142.233, 56.531, 156.864]
  Set speed (16.2 mm/s)
  Call Extruder(1290.61836)
  MoveL 7176 to (535.29, 543.72, 124) mm, rotated rx -180 ry 0 rz 160 deg; joints [10.828, 65.856, -15.62, -142.176, 56.684, 156.906]
  Set speed (16.2 mm/s)
  Call Extruder(1294.62600)
  MoveL 7177 to (534.39, 544.43, 124) mm, rotated rx -180 ry 0 rz 160 deg; joints [10.929, 65.712, -15.331, -142.123, 56.838, 156.951]
  Set speed (16.2 mm/s)
  Call Extruder(1298.51948)
  MoveL 7178 to (533.5, 545.11, 124) mm, rotated rx 180 ry 0 rz 160 deg; joints [11.025, 65.569, -15.046, -142.074, 56.988, 156.997]
  Set speed (16.2 mm/s)
  Call Extruder(1302.63728)
  MoveL 7179 to (532.55, 545.8, 124) mm, rotated rx -180 ry 0 rz 160 deg; joints [11.126, 65.416, -14.741, -142.024, 57.148, 157.049]
  Set speed (16.2 mm/s)
  Call Extruder(1306.65693)
  MoveL 7180 to (531.6, 546.46, 124) mm, rotated rx -180 ry 0 rz 160 deg; joints [11.223, 65.265, -14.437, -141.978, 57.305, 157.103]
  Set speed (16.2 mm/s)
  Call Extruder(1310.56814)
  MoveL 7181 to (530.67, 547.08, 124) mm, rotated rx 180 ry 0 rz 160 deg; joints [11.315, 65.115, -14.138, -141.936, 57.459, 157.158]
  Set speed (16.2 mm/s)
  Call Extruder(1314.56507)
  MoveL 7182 to (529.7, 547.7, 124) mm, rotated rx -180 ry 0 rz 160 deg; joints [11.408, 64.96, -13.827, -141.895, 57.617, 157.217]
  Set speed (16.2 mm/s)
  Call Extruder(1318.63429)
  MoveL 7183 to (528.71, 548.3, 124) mm, rotated rx 180 ry 0 rz 160 deg; joints [11.501, 64.8, -13.507, -141.856, 57.779, 157.28]
  Set speed (16.2 mm/s)
  Call Extruder(1322.59307)
  MoveL 7184 to (527.72, 548.87, 124) mm, rotated rx 180 ry 0 rz 160 deg; joints [11.59, 64.642, -13.191, -141.821, 57.938, 157.344]
  Set speed (16.2 mm/s)
  Call Extruder(1325.99511)
  MoveL 7185 to (526.87, 549.35, 124) mm, rotated rx 180 ry 0 rz 160 deg; joints [11.665, 64.506, -12.917, -141.793, 58.075, 157.401]
  Set speed (16.2 mm/s)
  Call Extruder(1332.07943)
  MoveL 7186 to (525.33, 550.16, 124) mm, rotated rx 180 ry 0 rz 160 deg; joints [11.795, 64.258, -12.421, -141.746, 58.32, 157.507]
  Set speed (16.2 mm/s)
  Call Extruder(1334.68312)
  MoveL 7187 to (524.66, 550.49, 124) mm, rotated rx 180 ry 0 rz 160 deg; joints [11.85, 64.151, -12.206, -141.728, 58.426, 157.555]
  Set speed (16.2 mm/s)
  Call Extruder(1338.79574)
  MoveL 7188 to (523.6, 550.99, 124) mm, rotated rx 180 ry 0 rz 160 deg; joints [11.935, 63.981, -11.863, -141.702, 58.593, 157.632]
  Set speed (16.2 mm/s)
  Call Extruder(1342.75425)
  MoveL 7189 to (522.56, 551.45, 124) mm, rotated rx -180 ry 0 rz 160 deg; joints [12.014, 63.814, -11.53, -141.68, 58.755, 157.709]
  Set speed (16.1 mm/s)
  Call Extruder(1346.65091)
  MoveL 7190 to (521.54, 551.89, 124) mm, rotated rx 180 ry 0 rz 160 deg; joints [12.09, 63.65, -11.2, -141.659, 58.913, 157.786]
  Set speed (16.2 mm/s)
  Call Extruder(1350.76738)
  MoveL 7191 to (520.44, 552.33, 124) mm, rotated rx 180 ry 0 rz 160 deg; joints [12.168, 63.475, -10.847, -141.64, 59.082, 157.871]
  Set speed (16.2 mm/s)
  Call Extruder(1354.67000)
  MoveL 7192 to (519.4, 552.73, 124) mm, rotated rx 180 ry 0 rz 160 deg; joints [12.242, 63.308, -10.512, -141.624, 59.242, 157.952]
  Set speed (16.2 mm/s)
  Call Extruder(1362.66407)
  MoveL 7193 to (517.24, 553.48, 124) mm, rotated rx -180 ry 0 rz 160 deg; joints [12.384, 62.962, -9.814, -141.599, 59.57, 158.127]
  Call Extruder(1370.65470)
  MoveL 7194 to (515.04, 554.14, 124) mm, rotated rx 180 ry 0 rz 160 deg; joints [12.518, 62.611, -9.108, -141.584, 59.899, 158.311]
  Set speed (16.2 mm/s)
  Call Extruder(1374.25156)
  MoveL 7195 to (514.05, 554.4, 124) mm, rotated rx -180 ry 0 rz 160 deg; joints [12.575, 62.452, -8.787, -141.581, 60.047, 158.396]
  Set speed (16.2 mm/s)
  Call Extruder(1378.80611)
  MoveL 7196 to (512.78, 554.71, 124) mm, rotated rx 180 ry 0 rz 160 deg; joints [12.646, 62.25, -8.38, -141.579, 60.233, 158.506]
  Set speed (16.2 mm/s)
  Call Extruder(1386.89476)
  MoveL 7197 to (510.51, 555.19, 124) mm, rotated rx -180 ry 0 rz 160 deg; joints [12.763, 61.889, -7.65, -141.583, 60.565, 158.707]
  Call Extruder(1394.97810)
  MoveL 7198 to (508.23, 555.58, 124) mm, rotated rx 180 ry 0 rz 160 deg; joints [12.871, 61.526, -6.915, -141.597, 60.895, 158.915]
  Set speed (16.2 mm/s)
  Call Extruder(1402.90458)
  MoveL 7199 to (505.98, 555.87, 124) mm, rotated rx -180 ry 0 rz 160 deg; joints [12.967, 61.167, -6.19, -141.621, 61.217, 159.126]
  Set speed (16.2 mm/s)
  Call Extruder(1410.96906)
  MoveL 7200 to (503.67, 556.07, 124) mm, rotated rx 180 ry 0 rz 160 deg; joints [13.054, 60.801, -5.449, -141.655, 61.542, 159.347]
  Set speed (16.2 mm/s)
  Call Extruder(1419.04431)
  MoveL 7201 to (501.36, 556.17, 124) mm, rotated rx 180 ry 0 rz 160 deg; joints [13.131, 60.434, -4.704, -141.699, 61.866, 159.574]
  Set speed (16.2 mm/s)
  Call Extruder(1426.96458)
  MoveL 7202 to (499.09, 556.18, 124) mm, rotated rx 180 ry 0 rz 160 deg; joints [13.197, 60.075, -3.973, -141.752, 62.18, 159.802]
  Set speed (10.0 mm/s)
  MoveL 7203 to (499.09, 556.18, 128) mm, rotated rx 180 ry 0 rz 160 deg; joints [13.197, 59.471, -3.759, -141.624, 61.875, 159.529]
  Set speed (120.0 mm/s)
  MoveL 7204 to (499.12, 554.25, 128) mm, rotated rx 180 ry 0 rz 160 deg; joints [12.962, 59.405, -3.625, -141.895, 61.846, 159.694]
  Set speed (16.3 mm/s)
  Call Extruder(1434.73048)
  MoveL 7205 to (496.89, 554.17, 128) mm, rotated rx 180 ry 0 rz 160 deg; joints [13.015, 59.049, -2.905, -141.958, 62.15, 159.921]
  Set speed (16.3 mm/s)
  Call Extruder(1442.45819)
  MoveL 7206 to (494.67, 554, 128) mm, rotated rx 180 ry 0 rz 160 deg; joints [13.057, 58.696, -2.191, -142.031, 62.45, 160.152]
  Call Extruder(1450.08835)
  MoveL 7207 to (492.49, 553.74, 128) mm, rotated rx -180 ry 0 rz 160 deg; joints [13.087, 58.349, -1.487, -142.112, 62.741, 160.384]
  Call Extruder(1457.75501)
  MoveL 7208 to (490.3, 553.39, 128) mm, rotated rx -180 ry 0 rz 160 deg; joints [13.106, 58.002, -0.783, -142.204, 63.029, 160.621]
  Set speed (16.3 mm/s)
  Call Extruder(1465.60608)
  MoveL 7209 to (488.09, 552.94, 128) mm, rotated rx 180 ry 0 rz 160 deg; joints [13.114, 57.649, -0.066, -142.308, 63.32, 160.867]
  Set speed (16.3 mm/s)
  Call Extruder(1469.39781)
  MoveL 7210 to (487.02, 552.68, 128) mm, rotated rx -180 ry 0 rz 160 deg; joints [13.114, 57.48, 0.278, -142.363, 63.458, 160.987]
  Set speed (16.2 mm/s)
  Call Extruder(1473.15111)
  MoveL 7211 to (485.98, 552.42, 128) mm, rotated rx 180 ry 0 rz 160 deg; joints [13.111, 57.313, 0.617, -142.418, 63.593, 161.105]
  Set speed (16.3 mm/s)
  Call Extruder(1480.82242)
  MoveL 7212 to (483.85, 551.81, 128) mm, rotated rx -180 ry 0 rz 160 deg; joints [13.096, 56.975, 1.306, -142.539, 63.867, 161.35]
  Call Extruder(1488.73892)
  MoveL 7213 to (481.69, 551.08, 128) mm, rotated rx -180 ry 0 rz 160 deg; joints [13.068, 56.629, 2.009, -142.675, 64.142, 161.605]
  Call Extruder(1496.54838)
  MoveL 7214 to (479.59, 550.28, 128) mm, rotated rx -180 ry 0 rz 160 deg; joints [13.028, 56.294, 2.694, -142.818, 64.408, 161.858]
  Set speed (16.3 mm/s)
  Call Extruder(1503.83602)
  MoveL 7215 to (477.66, 549.45, 128) mm, rotated rx 180 ry 0 rz 160 deg; joints [12.98, 55.985, 3.325, -142.962, 64.65, 162.095]
  Set speed (16.3 mm/s)
  Call Extruder(1509.57521)
  MoveL 7216 to (476.16, 548.75, 128) mm, rotated rx 180 ry 0 rz 160 deg; joints [12.934, 55.745, 3.816, -143.081, 64.836, 162.283]
  Set speed (16.3 mm/s)
  Call Extruder(1515.49223)
  MoveL 7217 to (474.64, 547.97, 128) mm, rotated rx -180 ry 0 rz 160 deg; joints [12.879, 55.501, 4.316, -143.211, 65.024, 162.477]
  Set speed (16.3 mm/s)
  Call Extruder(1519.32205)
  MoveL 7218 to (473.67, 547.45, 128) mm, rotated rx 180 ry 0 rz 160 deg; joints [12.84, 55.344, 4.636, -143.297, 65.144, 162.602]
  Set speed (16.3 mm/s)
  Call Extruder(1523.15014)
  MoveL 7219 to (472.71, 546.9, 128) mm, rotated rx 180 ry 0 rz 160 deg; joints [12.798, 55.19, 4.952, -143.386, 65.261, 162.727]
  Set speed (16.3 mm/s)
  Call Extruder(1527.07474)
  MoveL 7220 to (471.74, 546.32, 128) mm, rotated rx -180 ry 0 rz 160 deg; joints [12.752, 55.033, 5.274, -143.48, 65.38, 162.855]
  Set speed (16.3 mm/s)
  Call Extruder(1531.00073)
  MoveL 7221 to (470.78, 545.72, 128) mm, rotated rx 180 ry 0 rz 160 deg; joints [12.702, 54.878, 5.592, -143.577, 65.496, 162.984]
  Set speed (16.3 mm/s)
  Call Extruder(1534.84697)
  MoveL 7222 to (469.85, 545.12, 128) mm, rotated rx 180 ry 0 rz 160 deg; joints [12.65, 54.728, 5.899, -143.674, 65.608, 163.109]
  Set speed (16.3 mm/s)
  Call Extruder(1539.40810)
  MoveL 7223 to (468.77, 544.37, 128) mm, rotated rx 180 ry 0 rz 160 deg; joints [12.585, 54.553, 6.261, -143.792, 65.739, 163.258]
  Set speed (16.3 mm/s)
  Call Extruder(1542.50511)
  MoveL 7224 to (468.04, 543.85, 128) mm, rotated rx 180 ry 0 rz 160 deg; joints [12.538, 54.435, 6.503, -143.874, 65.826, 163.358]
  Set speed (16.3 mm/s)
  Call Extruder(1546.30608)
  MoveL 7225 to (467.16, 543.2, 128) mm, rotated rx -180 ry 0 rz 160 deg; joints [12.478, 54.292, 6.797, -143.977, 65.931, 163.482]
  Set speed (16.3 mm/s)
  Call Extruder(1550.14275)
  MoveL 7226 to (466.29, 542.52, 128) mm, rotated rx -180 ry 0 rz 160 deg; joints [12.415, 54.149, 7.09, -144.083, 66.035, 163.606]
  Set speed (16.3 mm/s)
  Call Extruder(1554.03447)
  MoveL 7227 to (465.42, 541.81, 128) mm, rotated rx -180 ry 0 rz 160 deg; joints [12.346, 54.007, 7.383, -144.194, 66.138, 163.731]
  Call Extruder(1557.97268)
  MoveL 7228 to (464.55, 541.08, 128) mm, rotated rx 180 ry 0 rz 160 deg; joints [12.275, 53.865, 7.676, -144.308, 66.24, 163.858]
  Set speed (16.3 mm/s)
  Call Extruder(1561.70662)
  MoveL 7229 to (463.74, 540.37, 128) mm, rotated rx -180 ry 0 rz 160 deg; joints [12.204, 53.732, 7.95, -144.418, 66.335, 163.978]
  Set speed (16.3 mm/s)
  Call Extruder(1567.48884)
  MoveL 7230 to (462.51, 539.24, 128) mm, rotated rx -180 ry 0 rz 160 deg; joints [12.089, 53.53, 8.366, -144.594, 66.478, 164.162]
  Call Extruder(1573.27593)
  MoveL 7231 to (461.33, 538.06, 128) mm, rotated rx -180 ry 0 rz 160 deg; joints [11.966, 53.334, 8.772, -144.775, 66.616, 164.345]
  Call Extruder(0.00000)
  Set speed (16.3 mm/s)
  Call Extruder(3.78521)
  MoveL 7232 to (460.57, 537.28, 128) mm, rotated rx -180 ry 0 rz 160 deg; joints [11.882, 53.208, 9.032, -144.896, 66.703, 164.464]
  Call Extruder(7.68309)
  MoveL 7233 to (459.81, 536.45, 128) mm, rotated rx -180 ry 0 rz 160 deg; joints [11.793, 53.081, 9.295, -145.023, 66.79, 164.586]
  Set speed (16.3 mm/s)
  Call Extruder(11.45557)
  MoveL 7234 to (459.09, 535.64, 128) mm, rotated rx 180 ry 0 rz 160 deg; joints [11.704, 52.96, 9.545, -145.148, 66.873, 164.703]
  Set speed (16.3 mm/s)
  Call Extruder(14.88391)
  MoveL 7235 to (458.44, 534.89, 128) mm, rotated rx -180 ry 0 rz 160 deg; joints [11.621, 52.852, 9.768, -145.264, 66.946, 164.809]
  Set speed (16.3 mm/s)
  Call Extruder(19.17858)
  MoveL 7236 to (457.66, 533.93, 128) mm, rotated rx -180 ry 0 rz 160 deg; joints [11.513, 52.72, 10.042, -145.411, 67.034, 164.94]
  Set speed (16.3 mm/s)
  Call Extruder(23.05888)
  MoveL 7237 to (456.97, 533.05, 128) mm, rotated rx 180 ry 0 rz 160 deg; joints [11.413, 52.603, 10.284, -145.546, 67.111, 165.059]
  Set speed (16.3 mm/s)
  Call Extruder(27.00970)
  MoveL 7238 to (456.28, 532.14, 128) mm, rotated rx -180 ry 0 rz 160 deg; joints [11.308, 52.487, 10.526, -145.685, 67.188, 165.178]
  Set speed (16.3 mm/s)
  Call Extruder(30.78094)
  MoveL 7239 to (455.65, 531.26, 128) mm, rotated rx 180 ry 0 rz 160 deg; joints [11.205, 52.378, 10.751, -145.821, 67.258, 165.291]
  Call Extruder(34.61109)
  MoveL 7240 to (455.02, 530.35, 128) mm, rotated rx -180 ry 0 rz 160 deg; joints [11.098, 52.271, 10.974, -145.96, 67.327, 165.404]
  Call Extruder(38.47057)
  MoveL 7241 to (454.41, 529.42, 128) mm, rotated rx -180 ry 0 rz 160 deg; joints [10.988, 52.165, 11.194, -146.103, 67.393, 165.518]
  Set speed (16.3 mm/s)
  Call Extruder(42.28958)
  MoveL 7242 to (453.82, 528.49, 128) mm, rotated rx 180 ry 0 rz 160 deg; joints [10.876, 52.063, 11.406, -146.246, 67.457, 165.629]
  Call Extruder(46.25287)
  MoveL 7243 to (453.23, 527.51, 128) mm, rotated rx 180 ry 0 rz 160 deg; joints [10.757, 51.96, 11.62, -146.396, 67.52, 165.744]
  Set speed (16.3 mm/s)
  Call Extruder(50.03231)
  MoveL 7244 to (452.69, 526.57, 128) mm, rotated rx 180 ry 0 rz 160 deg; joints [10.641, 51.864, 11.818, -146.541, 67.577, 165.852]
  Set speed (16.3 mm/s)
  Call Extruder(53.82057)
  MoveL 7245 to (452.16, 525.61, 128) mm, rotated rx 180 ry 0 rz 160 deg; joints [10.523, 51.771, 12.012, -146.688, 67.632, 165.959]
  Set speed (16.3 mm/s)
  Call Extruder(57.68064)
  MoveL 7246 to (451.65, 524.63, 128) mm, rotated rx -180 ry 0 rz 160 deg; joints [10.4, 51.679, 12.204, -146.839, 67.686, 166.067]
  Call Extruder(61.71069)
  MoveL 7247 to (451.13, 523.59, 128) mm, rotated rx -180 ry 0 rz 160 deg; joints [10.269, 51.586, 12.397, -146.999, 67.739, 166.178]
  Set speed (16.3 mm/s)
  Call Extruder(69.38248)
  MoveL 7248 to (450.21, 521.58, 128) mm, rotated rx 180 ry 0 rz 160 deg; joints [10.013, 51.418, 12.748, -147.308, 67.831, 166.387]
  Set speed (16.3 mm/s)
  Call Extruder(76.84750)
  MoveL 7249 to (449.4, 519.58, 128) mm, rotated rx -180 ry 0 rz 160 deg; joints [9.755, 51.266, 13.065, -147.615, 67.91, 166.585]
  Set speed (16.2 mm/s)
  Call Extruder(79.00392)
  MoveL 7250 to (449.17, 519, 128) mm, rotated rx -180 ry 0 rz 160 deg; joints [9.679, 51.224, 13.152, -147.704, 67.931, 166.641]
  Call Extruder(84.91392)
  MoveL 7251 to (448.6, 517.4, 128) mm, rotated rx 180 ry 0 rz 160 deg; joints [9.469, 51.114, 13.382, -147.951, 67.984, 166.792]
  Set speed (16.3 mm/s)
  Call Extruder(92.25623)
  MoveL 7252 to (447.96, 515.38, 128) mm, rotated rx 180 ry 0 rz 160 deg; joints [9.2, 50.988, 13.646, -148.262, 68.04, 166.976]
  Set speed (16.3 mm/s)
  Call Extruder(96.34753)
  MoveL 7253 to (447.65, 514.25, 128) mm, rotated rx -180 ry 0 rz 160 deg; joints [9.048, 50.923, 13.782, -148.438, 68.066, 167.076]
  Set speed (16.3 mm/s)
  Call Extruder(100.02660)
  MoveL 7254 to (447.38, 513.23, 128) mm, rotated rx -180 ry 0 rz 160 deg; joints [8.91, 50.866, 13.9, -148.596, 68.087, 167.165]
  Set speed (16.2 mm/s)
  Call Extruder(103.39781)
  MoveL 7255 to (447.15, 512.28, 128) mm, rotated rx 180 ry 0 rz 160 deg; joints [8.781, 50.818, 14.001, -148.742, 68.104, 167.245]
  Set speed (16.2 mm/s)
  Call Extruder(108.64629)
  MoveL 7256 to (446.82, 510.81, 128) mm, rotated rx 180 ry 0 rz 160 deg; joints [8.58, 50.746, 14.15, -148.969, 68.127, 167.367]
  Set speed (16.3 mm/s)
  Call Extruder(115.62909)
  MoveL 7257 to (446.46, 508.83, 128) mm, rotated rx 180 ry 0 rz 160 deg; joints [8.307, 50.661, 14.328, -149.275, 68.147, 167.525]
  Set speed (16.3 mm/s)
  Call Extruder(123.34772)
  MoveL 7258 to (446.14, 506.63, 128) mm, rotated rx 180 ry 0 rz 160 deg; joints [8.001, 50.579, 14.5, -149.616, 68.159, 167.694]
  Call Extruder(131.03759)
  MoveL 7259 to (445.92, 504.42, 128) mm, rotated rx 180 ry 0 rz 160 deg; joints [7.692, 50.511, 14.643, -149.956, 68.158, 167.856]
  Set speed (16.3 mm/s)
  Call Extruder(138.54756)
  MoveL 7260 to (445.78, 502.26, 128) mm, rotated rx 180 ry 0 rz 160 deg; joints [7.387, 50.457, 14.757, -150.29, 68.145, 168.008]
  Call Extruder(146.68655)
  MoveL 7261 to (445.74, 499.91, 128) mm, rotated rx 180 ry 0 rz 160 deg; joints [7.053, 50.413, 14.849, -150.652, 68.119, 168.165]
  Set speed (16.3 mm/s)
  Call Extruder(153.36031)
  MoveL 7262 to (445.77, 497.99, 128) mm, rotated rx -180 ry 0 rz 160 deg; joints [6.777, 50.387, 14.903, -150.948, 68.087, 168.288]
  Set speed (16.3 mm/s)
  Call Extruder(160.19389)
  MoveL 7263 to (445.88, 496.02, 128) mm, rotated rx -180 ry 0 rz 160 deg; joints [6.494, 50.372, 14.935, -151.25, 68.044, 168.408]
  Set speed (16.3 mm/s)
  Call Extruder(167.13853)
  MoveL 7264 to (446.07, 494.03, 128) mm, rotated rx 180 ry 0 rz 160 deg; joints [6.206, 50.367, 14.946, -151.556, 67.992, 168.525]
  Call Extruder(174.05539)
  MoveL 7265 to (446.32, 492.05, 128) mm, rotated rx 180 ry 0 rz 160 deg; joints [5.919, 50.372, 14.934, -151.858, 67.929, 168.636]
  Call Extruder(181.08849)
  MoveL 7266 to (446.66, 490.05, 128) mm, rotated rx -180 ry 0 rz 160 deg; joints [5.627, 50.39, 14.898, -152.163, 67.855, 168.742]
  Set speed (16.3 mm/s)
  Call Extruder(187.85950)
  MoveL 7267 to (447.05, 488.14, 128) mm, rotated rx 180 ry 0 rz 160 deg; joints [5.348, 50.417, 14.841, -152.453, 67.775, 168.839]
  Set speed (16.3 mm/s)
  Call Extruder(194.85231)
  MoveL 7268 to (447.53, 486.19, 128) mm, rotated rx 180 ry 0 rz 160 deg; joints [5.061, 50.455, 14.76, -152.749, 67.682, 168.933]
  Set speed (16.3 mm/s)
  Call Extruder(201.68760)
  MoveL 7269 to (448.06, 484.29, 128) mm, rotated rx 180 ry 0 rz 160 deg; joints [4.783, 50.504, 14.658, -153.035, 67.581, 169.019]
  Set speed (16.3 mm/s)
  Call Extruder(208.73014)
  MoveL 7270 to (448.69, 482.36, 128) mm, rotated rx -180 ry 0 rz 160 deg; joints [4.499, 50.564, 14.531, -153.324, 67.468, 169.102]
  Set speed (16.3 mm/s)
  Call Extruder(215.74012)
  MoveL 7271 to (449.38, 480.46, 128) mm, rotated rx 180 ry 0 rz 160 deg; joints [4.22, 50.636, 14.382, -153.606, 67.346, 169.179]
  Call Extruder(222.40021)
  MoveL 7272 to (450.1, 478.68, 128) mm, rotated rx -180 ry 0 rz 160 deg; joints [3.959, 50.714, 14.219, -153.869, 67.221, 169.245]
  Set speed (16.3 mm/s)
  Call Extruder(229.44157)
  MoveL 7273 to (450.93, 476.83, 128) mm, rotated rx -180 ry 0 rz 160 deg; joints [3.687, 50.806, 14.025, -154.14, 67.079, 169.31]
  Set speed (16.3 mm/s)
  Call Extruder(236.54367)
  MoveL 7274 to (451.84, 475, 128) mm, rotated rx 180 ry 0 rz 160 deg; joints [3.418, 50.91, 13.807, -154.406, 66.927, 169.368]
  Set speed (16.3 mm/s)
  Call Extruder(243.28344)
  MoveL 7275 to (452.77, 473.29, 128) mm, rotated rx -180 ry 0 rz 160 deg; joints [3.167, 51.019, 13.58, -154.652, 66.774, 169.418]
  Call Extruder(250.24440)
  MoveL 7276 to (453.79, 471.56, 128) mm, rotated rx 180 ry 0 rz 160 deg; joints [2.915, 51.142, 13.324, -154.898, 66.607, 169.463]
  Set speed (16.3 mm/s)
  Call Extruder(257.25166)
  MoveL 7277 to (454.88, 469.86, 128) mm, rotated rx -180 ry 0 rz 160 deg; joints [2.666, 51.275, 13.046, -155.138, 66.43, 169.503]
  Set speed (16.3 mm/s)
  Call Extruder(264.16959)
  MoveL 7278 to (456.01, 468.23, 128) mm, rotated rx -180 ry 0 rz 160 deg; joints [2.428, 51.417, 12.751, -155.366, 66.248, 169.535]
  Set speed (16.3 mm/s)
  Call Extruder(271.14742)
  MoveL 7279 to (457.22, 466.62, 128) mm, rotated rx -180 ry 0 rz 160 deg; joints [2.194, 51.569, 12.433, -155.587, 66.055, 169.562]
  Set speed (16.3 mm/s)
  Call Extruder(277.95906)
  MoveL 7280 to (458.46, 465.09, 128) mm, rotated rx 180 ry 0 rz 160 deg; joints [1.973, 51.727, 12.104, -155.793, 65.859, 169.582]
  Set speed (16.3 mm/s)
  Call Extruder(285.00363)
  MoveL 7281 to (459.8, 463.56, 128) mm, rotated rx 180 ry 0 rz 160 deg; joints [1.753, 51.9, 11.744, -155.996, 65.649, 169.596]
  Call Extruder(291.98629)
  MoveL 7282 to (461.17, 462.09, 128) mm, rotated rx -180 ry 0 rz 160 deg; joints [1.542, 52.08, 11.369, -156.188, 65.433, 169.603]
  Call Extruder(298.68847)
  MoveL 7283 to (462.55, 460.74, 128) mm, rotated rx -180 ry 0 rz 160 deg; joints [1.348, 52.262, 10.992, -156.362, 65.219, 169.604]
  Call Extruder(305.74755)
  MoveL 7284 to (464.05, 459.36, 128) mm, rotated rx -180 ry 0 rz 160 deg; joints [1.153, 52.462, 10.577, -156.534, 64.986, 169.599]
  Set speed (16.3 mm/s)
  Call Extruder(312.77245)
  MoveL 7285 to (465.59, 458.05, 128) mm, rotated rx 180 ry 0 rz 160 deg; joints [0.967, 52.67, 10.147, -156.694, 64.748, 169.587]
  Call Extruder(320.06349)
  MoveL 7286 to (467.24, 456.75, 128) mm, rotated rx -180 ry 0 rz 160 deg; joints [0.784, 52.894, 9.682, -156.848, 64.494, 169.567]
  Set speed (16.3 mm/s)
  Call Extruder(325.97204)
  MoveL 7287 to (468.61, 455.74, 128) mm, rotated rx 180 ry 0 rz 160 deg; joints [0.644, 53.082, 9.293, -156.964, 64.284, 169.546]
  Set speed (16.3 mm/s)
  Call Extruder(333.48176)
  MoveL 7288 to (470.4, 454.52, 128) mm, rotated rx -180 ry 0 rz 160 deg; joints [0.475, 53.329, 8.782, -157.098, 64.01, 169.512]
  Set speed (16.3 mm/s)
  Call Extruder(340.33932)
  MoveL 7289 to (472.08, 453.48, 128) mm, rotated rx 180 ry 0 rz 160 deg; joints [0.331, 53.563, 8.3, -157.209, 63.755, 169.474]
  Call Extruder(347.42707)
  MoveL 7290 to (473.85, 452.45, 128) mm, rotated rx 180 ry 0 rz 160 deg; joints [0.191, 53.811, 7.787, -157.311, 63.486, 169.428]
  Set speed (16.2 mm/s)
  Call Extruder(355.24721)
  MoveL 7291 to (475.84, 451.41, 128) mm, rotated rx 180 ry 0 rz 160 deg; joints [0.05, 54.093, 7.206, -157.409, 63.184, 169.369]
  Set speed (16.2 mm/s)
  Call Extruder(361.25880)
  MoveL 7292 to (477.4, 450.67, 128) mm, rotated rx -180 ry 0 rz 160 deg; joints [-0.05, 54.316, 6.748, -157.474, 62.948, 169.318]
  Set speed (16.3 mm/s)
  Call Extruder(368.23146)
  MoveL 7293 to (479.25, 449.86, 128) mm, rotated rx 180 ry 0 rz 160 deg; joints [-0.158, 54.58, 6.205, -157.537, 62.67, 169.252]
  Set speed (16.3 mm/s)
  Call Extruder(375.08238)
  MoveL 7294 to (481.09, 449.14, 128) mm, rotated rx 180 ry 0 rz 160 deg; joints [-0.253, 54.845, 5.659, -157.588, 62.393, 169.18]
  Set speed (16.3 mm/s)
  Call Extruder(381.83691)
  MoveL 7295 to (482.92, 448.5, 128) mm, rotated rx 180 ry 0 rz 160 deg; joints [-0.338, 55.112, 5.111, -157.625, 62.118, 169.103]
  Set speed (16.3 mm/s)
  Call Extruder(388.98623)
  MoveL 7296 to (484.89, 447.89, 128) mm, rotated rx 180 ry 0 rz 160 deg; joints [-0.417, 55.401, 4.52, -157.651, 61.823, 169.014]
  Set speed (16.3 mm/s)
  Call Extruder(395.91500)
  MoveL 7297 to (486.82, 447.36, 128) mm, rotated rx 180 ry 0 rz 160 deg; joints [-0.483, 55.685, 3.938, -157.665, 61.535, 168.92]
  Call Extruder(402.84275)
  MoveL 7298 to (488.76, 446.92, 128) mm, rotated rx 180 ry 0 rz 160 deg; joints [-0.54, 55.974, 3.347, -157.665, 61.244, 168.82]
  Set speed (16.3 mm/s)
  Call Extruder(409.64592)
  MoveL 7299 to (490.69, 446.54, 128) mm, rotated rx -180 ry 0 rz 160 deg; joints [-0.586, 56.262, 2.759, -157.654, 60.957, 168.714]
  Call Extruder(416.32226)
  MoveL 7300 to (492.59, 446.25, 128) mm, rotated rx -180 ry 0 rz 160 deg; joints [-0.622, 56.548, 2.174, -157.631, 60.674, 168.604]
  Set speed (16.3 mm/s)
  Call Extruder(423.59050)
  MoveL 7301 to (494.67, 446, 128) mm, rotated rx -180 ry 0 rz 160 deg; joints [-0.651, 56.864, 1.53, -157.593, 60.366, 168.477]
  Set speed (16.3 mm/s)
  Call Extruder(430.42426)
  MoveL 7302 to (496.63, 445.84, 128) mm, rotated rx -180 ry 0 rz 160 deg; joints [-0.668, 57.164, 0.919, -157.545, 60.074, 168.35]
  Set speed (16.3 mm/s)
  Call Extruder(437.55212)
  MoveL 7303 to (498.68, 445.75, 128) mm, rotated rx 180 ry 0 rz 160 deg; joints [-0.676, 57.481, 0.275, -157.481, 59.77, 168.21]
  Set speed (16.3 mm/s)
  Call Extruder(444.39816)
  MoveL 7304 to (500.66, 445.74, 128) mm, rotated rx -180 ry 0 rz 160 deg; joints [-0.675, 57.787, -0.347, -157.409, 59.478, 168.068]
  Set speed (16.3 mm/s)
  Call Extruder(451.40069)
  MoveL 7305 to (502.68, 445.8, 128) mm, rotated rx -180 ry 0 rz 160 deg; joints [-0.664, 58.103, -0.989, -157.322, 59.18, 167.916]
  Call Extruder(458.24604)
  MoveL 7306 to (504.65, 445.94, 128) mm, rotated rx 180 ry 0 rz 160 deg; joints [-0.645, 58.414, -1.619, -157.226, 58.89, 167.761]
  Set speed (16.3 mm/s)
  Call Extruder(465.25800)
  MoveL 7307 to (506.66, 446.15, 128) mm, rotated rx 180 ry 0 rz 160 deg; joints [-0.615, 58.733, -2.266, -157.115, 58.594, 167.595]
  Set speed (16.3 mm/s)
  Call Extruder(471.99485)
  MoveL 7308 to (508.58, 446.42, 128) mm, rotated rx -180 ry 0 rz 160 deg; joints [-0.578, 59.041, -2.889, -156.997, 58.312, 167.429]
  Set speed (16.3 mm/s)
  Call Extruder(479.02324)
  MoveL 7309 to (510.57, 446.78, 128) mm, rotated rx 180 ry 0 rz 160 deg; joints [-0.531, 59.363, -3.541, -156.863, 58.019, 167.248]
  Set speed (16.3 mm/s)
  Call Extruder(485.34673)
  MoveL 7310 to (512.35, 447.16, 128) mm, rotated rx 180 ry 0 rz 160 deg; joints [-0.482, 59.653, -4.126, -156.733, 57.758, 167.08]
  Set speed (16.3 mm/s)
  Call Extruder(492.80207)
  MoveL 7311 to (514.43, 447.69, 128) mm, rotated rx 180 ry 0 rz 160 deg; joints [-0.414, 59.995, -4.816, -156.567, 57.454, 166.875]
  Set speed (16.3 mm/s)
  Call Extruder(499.84470)
  MoveL 7312 to (516.38, 448.27, 128) mm, rotated rx 180 ry 0 rz 160 deg; joints [-0.341, 60.318, -5.467, -156.399, 57.17, 166.674]
  Set speed (16.3 mm/s)
  Call Extruder(506.83085)
  MoveL 7313 to (518.29, 448.91, 128) mm, rotated rx 180 ry 0 rz 160 deg; joints [-0.261, 60.637, -6.11, -156.222, 56.892, 166.468]
  Call Extruder(513.67321)
  MoveL 7314 to (520.14, 449.61, 128) mm, rotated rx -180 ry 0 rz 160 deg; joints [-0.175, 60.949, -6.737, -156.038, 56.624, 166.261]
  Call Extruder(520.68692)
  MoveL 7315 to (522, 450.4, 128) mm, rotated rx 180 ry 0 rz 160 deg; joints [-0.078, 61.266, -7.375, -155.839, 56.354, 166.042]
  Set speed (16.3 mm/s)
  Call Extruder(527.63077)
  MoveL 7316 to (523.81, 451.24, 128) mm, rotated rx 180 ry 0 rz 160 deg; joints [0.024, 61.578, -8.002, -155.633, 56.092, 165.82]
  Call Extruder(534.46671)
  MoveL 7317 to (525.57, 452.14, 128) mm, rotated rx -180 ry 0 rz 160 deg; joints [0.132, 61.883, -8.613, -155.421, 55.84, 165.596]
  Set speed (16.3 mm/s)
  Call Extruder(541.48677)
  MoveL 7318 to (527.33, 453.13, 128) mm, rotated rx -180 ry 0 rz 160 deg; joints [0.25, 62.193, -9.235, -155.194, 55.586, 165.36]
  Set speed (16.3 mm/s)
  Call Extruder(548.41414)
  MoveL 7319 to (529.04, 454.17, 128) mm, rotated rx 180 ry 0 rz 160 deg; joints [0.374, 62.495, -9.841, -154.96, 55.343, 165.123]
  Set speed (16.3 mm/s)
  Call Extruder(555.13067)
  MoveL 7320 to (530.66, 455.23, 128) mm, rotated rx 180 ry 0 rz 160 deg; joints [0.5, 62.785, -10.421, -154.727, 55.112, 164.888]
  Set speed (16.3 mm/s)
  Call Extruder(562.10323)
  MoveL 7321 to (532.29, 456.4, 128) mm, rotated rx 180 ry 0 rz 160 deg; joints [0.637, 63.081, -11.013, -154.476, 54.881, 164.64]
  Call Extruder(569.30124)
  MoveL 7322 to (533.94, 457.66, 128) mm, rotated rx 180 ry 0 rz 160 deg; joints [0.785, 63.383, -11.615, -154.21, 54.649, 164.38]
  Set speed (16.3 mm/s)
  Call Extruder(576.08257)
  MoveL 7323 to (535.44, 458.92, 128) mm, rotated rx -180 ry 0 rz 160 deg; joints [0.93, 63.661, -12.171, -153.951, 54.439, 164.132]
  Set speed (16.3 mm/s)
  Call Extruder(583.06913)
  MoveL 7324 to (536.94, 460.26, 128) mm, rotated rx -180 ry 0 rz 160 deg; joints [1.086, 63.942, -12.733, -153.679, 54.23, 163.872]
  Call Extruder(589.94292)
  MoveL 7325 to (538.37, 461.63, 128) mm, rotated rx 180 ry 0 rz 160 deg; joints [1.244, 64.213, -13.273, -153.405, 54.034, 163.614]
  Set speed (16.3 mm/s)
  Call Extruder(593.70148)
  MoveL 7326 to (539.13, 462.41, 128) mm, rotated rx -180 ry 0 rz 160 deg; joints [1.333, 64.358, -13.561, -153.252, 53.93, 163.473]
  Call Extruder(597.62312)
  MoveL 7327 to (539.9, 463.23, 128) mm, rotated rx -180 ry 0 rz 160 deg; joints [1.427, 64.508, -13.86, -153.092, 53.824, 163.324]
  Call Extruder(601.39138)
  MoveL 7328 to (540.63, 464.04, 128) mm, rotated rx 180 ry 0 rz 160 deg; joints [1.519, 64.649, -14.141, -152.936, 53.726, 163.18]
  Set speed (16.3 mm/s)
  Call Extruder(605.27326)
  MoveL 7329 to (541.36, 464.88, 128) mm, rotated rx -180 ry 0 rz 160 deg; joints [1.616, 64.792, -14.427, -152.774, 53.628, 163.032]
  Set speed (16.3 mm/s)
  Call Extruder(609.19393)
  MoveL 7330 to (542.09, 465.75, 128) mm, rotated rx 180 ry 0 rz 160 deg; joints [1.714, 64.935, -14.711, -152.608, 53.531, 162.882]
  Set speed (16.3 mm/s)
  Call Extruder(612.91742)
  MoveL 7331 to (542.76, 466.59, 128) mm, rotated rx 180 ry 0 rz 160 deg; joints [1.81, 65.068, -14.976, -152.45, 53.442, 162.739]
  Set speed (16.3 mm/s)
  Call Extruder(616.80875)
  MoveL 7332 to (543.44, 467.48, 128) mm, rotated rx 180 ry 0 rz 160 deg; joints [1.911, 65.205, -15.247, -152.283, 53.353, 162.589]
  Set speed (16.3 mm/s)
  Call Extruder(620.61269)
  MoveL 7333 to (544.09, 468.36, 128) mm, rotated rx 180 ry 0 rz 160 deg; joints [2.011, 65.336, -15.508, -152.119, 53.268, 162.442]
  Call Extruder(624.48584)
  MoveL 7334 to (544.73, 469.28, 128) mm, rotated rx 180 ry 0 rz 160 deg; joints [2.114, 65.466, -15.767, -151.951, 53.186, 162.293]
  Call Extruder(628.34654)
  MoveL 7335 to (545.35, 470.2, 128) mm, rotated rx 180 ry 0 rz 160 deg; joints [2.218, 65.594, -16.021, -151.783, 53.106, 162.145]
  Set speed (16.3 mm/s)
  Call Extruder(633.09430)
  MoveL 7336 to (546.09, 471.36, 128) mm, rotated rx -180 ry 0 rz 160 deg; joints [2.348, 65.747, -16.326, -151.574, 53.013, 161.962]
  Set speed (16.3 mm/s)
  Call Extruder(639.96905)
  MoveL 7337 to (547.1, 473.06, 128) mm, rotated rx -180 ry 0 rz 160 deg; joints [2.54, 65.961, -16.751, -151.27, 52.888, 161.698]
  Set speed (16.3 mm/s)
  Call Extruder(643.79527)
  MoveL 7338 to (547.64, 474.02, 128) mm, rotated rx 180 ry 0 rz 160 deg; joints [2.648, 66.076, -16.978, -151.1, 52.823, 161.552]
  Set speed (16.3 mm/s)
  Call Extruder(647.62019)
  MoveL 7339 to (548.16, 475, 128) mm, rotated rx -180 ry 0 rz 160 deg; joints [2.757, 66.188, -17.2, -150.93, 52.761, 161.407]
  Set speed (16.3 mm/s)
  Call Extruder(651.39202)
  MoveL 7340 to (548.65, 475.97, 128) mm, rotated rx 180 ry 0 rz 160 deg; joints [2.865, 66.295, -17.413, -150.761, 52.704, 161.264]
  Set speed (16.3 mm/s)
  Call Extruder(655.48088)
  MoveL 7341 to (549.16, 477.03, 128) mm, rotated rx 180 ry 0 rz 160 deg; joints [2.984, 66.408, -17.637, -150.578, 52.645, 161.11]
  Call Extruder(659.26176)
  MoveL 7342 to (549.61, 478.02, 128) mm, rotated rx -180 ry 0 rz 160 deg; joints [3.095, 66.509, -17.837, -150.409, 52.595, 160.968]
  Set speed (16.3 mm/s)
  Call Extruder(666.80566)
  MoveL 7343 to (550.45, 480.03, 128) mm, rotated rx -180 ry 0 rz 160 deg; joints [3.319, 66.701, -18.218, -150.071, 52.505, 160.688]
  Call Extruder(674.46664)
  MoveL 7344 to (551.22, 482.1, 128) mm, rotated rx 180 ry 0 rz 160 deg; joints [3.55, 66.882, -18.577, -149.727, 52.428, 160.408]
  Set speed (16.3 mm/s)
  Call Extruder(682.21582)
  MoveL 7345 to (551.92, 484.22, 128) mm, rotated rx -180 ry 0 rz 160 deg; joints [3.787, 67.051, -18.911, -149.381, 52.365, 160.131]
  Set speed (16.2 mm/s)
  Call Extruder(686.15490)
  MoveL 7346 to (552.23, 485.31, 128) mm, rotated rx 180 ry 0 rz 160 deg; joints [3.909, 67.13, -19.068, -149.207, 52.34, 159.992]
  Set speed (16.2 mm/s)
  Call Extruder(690.00511)
  MoveL 7347 to (552.52, 486.38, 128) mm, rotated rx -180 ry 0 rz 160 deg; joints [4.028, 67.206, -19.218, -149.036, 52.317, 159.858]
  Set speed (16.3 mm/s)
  Call Extruder(697.67685)
  MoveL 7348 to (553.04, 488.53, 128) mm, rotated rx -180 ry 0 rz 160 deg; joints [4.268, 67.343, -19.49, -148.698, 52.285, 159.596]
  Call Extruder(705.20474)
  MoveL 7349 to (553.45, 490.66, 128) mm, rotated rx -180 ry 0 rz 160 deg; joints [4.505, 67.463, -19.726, -148.369, 52.269, 159.347]
  Set speed (16.3 mm/s)
  Call Extruder(713.09735)
  MoveL 7350 to (553.8, 492.91, 128) mm, rotated rx -180 ry 0 rz 160 deg; joints [4.757, 67.572, -19.942, -148.028, 52.267, 159.094]
  Set speed (16.3 mm/s)
  Call Extruder(720.90060)
  MoveL 7351 to (554.04, 495.14, 128) mm, rotated rx 180 ry 0 rz 160 deg; joints [5.007, 67.663, -20.122, -147.696, 52.281, 158.853]
  Set speed (16.3 mm/s)
  Call Extruder(728.49336)
  MoveL 7352 to (554.2, 497.32, 128) mm, rotated rx 180 ry 0 rz 160 deg; joints [5.252, 67.736, -20.266, -147.378, 52.31, 158.628]
  Set speed (16.3 mm/s)
  Call Extruder(736.19422)
  MoveL 7353 to (554.26, 499.54, 128) mm, rotated rx 180 ry 0 rz 160 deg; joints [5.502, 67.793, -20.379, -147.061, 52.355, 158.411]
  Set speed (16.3 mm/s)
  Call Extruder(743.74472)
  MoveL 7354 to (554.23, 501.72, 128) mm, rotated rx -180 ry 0 rz 160 deg; joints [5.747, 67.832, -20.456, -146.757, 52.414, 158.209]
  Set speed (16.3 mm/s)
  Call Extruder(751.57540)
  MoveL 7355 to (554.12, 503.98, 128) mm, rotated rx -180 ry 0 rz 160 deg; joints [6.003, 67.856, -20.503, -146.449, 52.49, 158.011]
  Set speed (16.3 mm/s)
  Call Extruder(759.18459)
  MoveL 7356 to (553.91, 506.16, 128) mm, rotated rx -180 ry 0 rz 160 deg; joints [6.251, 67.861, -20.515, -146.156, 52.578, 157.83]
  Set speed (16.3 mm/s)
  Call Extruder(767.08075)
  MoveL 7357 to (553.61, 508.42, 128) mm, rotated rx -180 ry 0 rz 160 deg; joints [6.509, 67.851, -20.494, -145.861, 52.684, 157.655]
  Call Extruder(774.65707)
  MoveL 7358 to (553.22, 510.57, 128) mm, rotated rx 180 ry 0 rz 160 deg; joints [6.755, 67.823, -20.439, -145.586, 52.801, 157.501]
  Set speed (16.3 mm/s)
  Call Extruder(782.43873)
  MoveL 7359 to (552.74, 512.76, 128) mm, rotated rx 180 ry 0 rz 160 deg; joints [7.008, 67.777, -20.348, -145.312, 52.935, 157.356]
  Set speed (16.3 mm/s)
  Call Extruder(786.26316)
  MoveL 7360 to (552.47, 513.83, 128) mm, rotated rx 180 ry 0 rz 160 deg; joints [7.132, 67.748, -20.29, -145.181, 53.006, 157.29]
  Call Extruder(790.29454)
